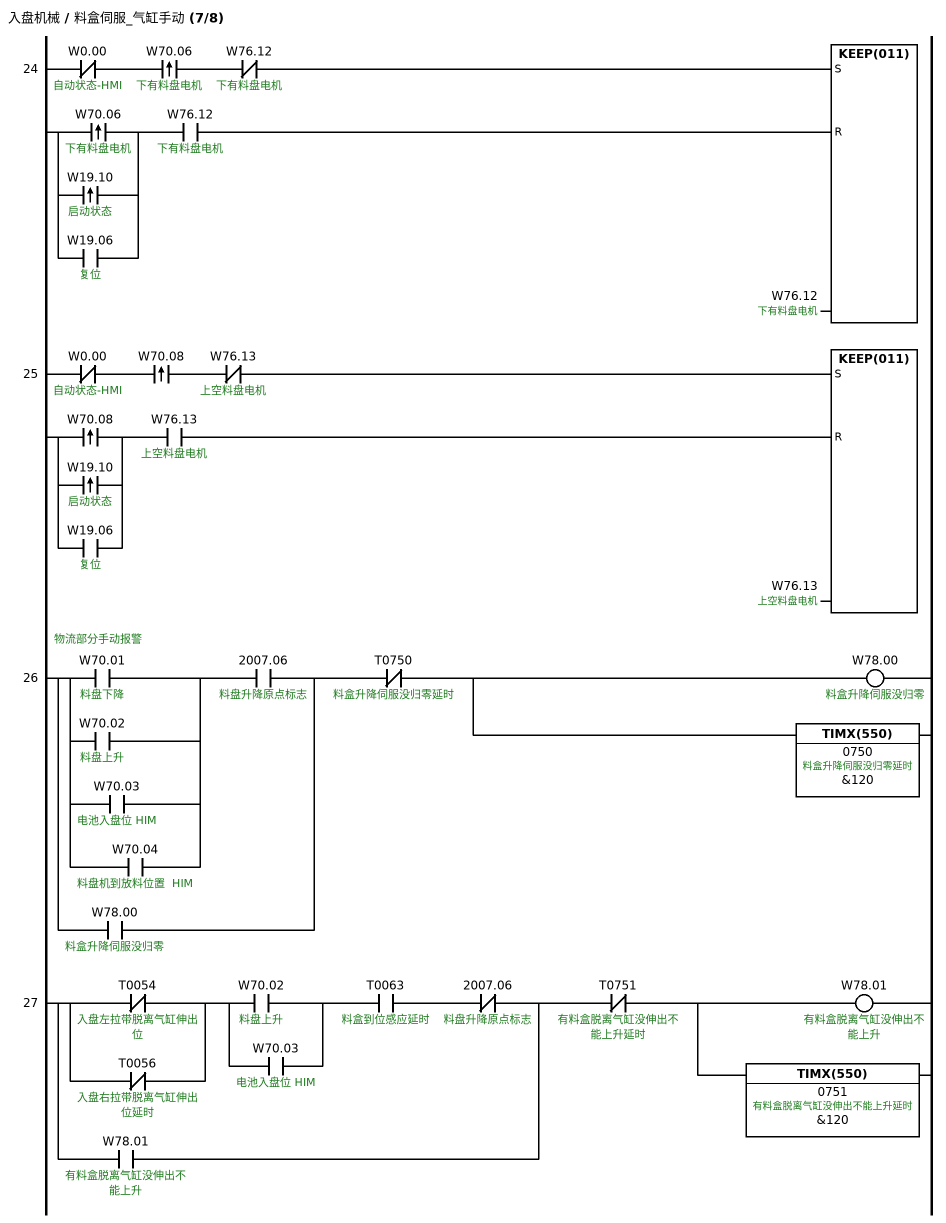
; [picture p216: 入盘机械 / 料盒伺服_气缸手动, rungs 24-27]
; rung 24
LDNOT W0.00  ; 自动状态-HMI
@AND W70.06  ; 下有料盘电机
ANDNOT W76.12  ; 下有料盘电机
@LD W70.06  ; 下有料盘电机
@OR W19.10  ; 启动状态
OR W19.06  ; 复位
AND W76.12  ; 下有料盘电机
KEEP(011) W76.12  ; 下有料盘电机
; rung 25
LDNOT W0.00  ; 自动状态-HMI
@AND W70.08
ANDNOT W76.13  ; 上空料盘电机
@LD W70.08
@OR W19.10  ; 启动状态
OR W19.06  ; 复位
AND W76.13  ; 上空料盘电机
KEEP(011) W76.13  ; 上空料盘电机
; rung 26: 物流部分手动报警
LD W70.01  ; 料盘下降
OR W70.02  ; 料盘上升
OR W70.03  ; 电池入盘位 HIM
OR W70.04  ; 料盘机到放料位置  HIM
AND 2007.06  ; 料盘升降原点标志
OR W78.00  ; 料盒升降伺服没归零
ANDNOT T0750  ; 料盒升降伺服没归零延时
OUT W78.00  ; 料盒升降伺服没归零
TIMX(550) 0750 &120  ; 料盒升降伺服没归零延时
; rung 27
LDNOT T0054  ; 入盘左拉带脱离气缸伸出位
ORNOT T0056  ; 入盘右拉带脱离气缸伸出位延时
LD W70.02  ; 料盘上升
OR W70.03  ; 电池入盘位 HIM
ANDLD
AND T0063  ; 料盒到位感应延时
ANDNOT 2007.06  ; 料盘升降原点标志
OR W78.01  ; 有料盒脱离气缸没伸出不能上升
ANDNOT T0751  ; 有料盒脱离气缸没伸出不能上升延时
OUT W78.01  ; 有料盒脱离气缸没伸出不能上升
TIMX(550) 0751 &120  ; 有料盒脱离气缸没伸出不能上升延时

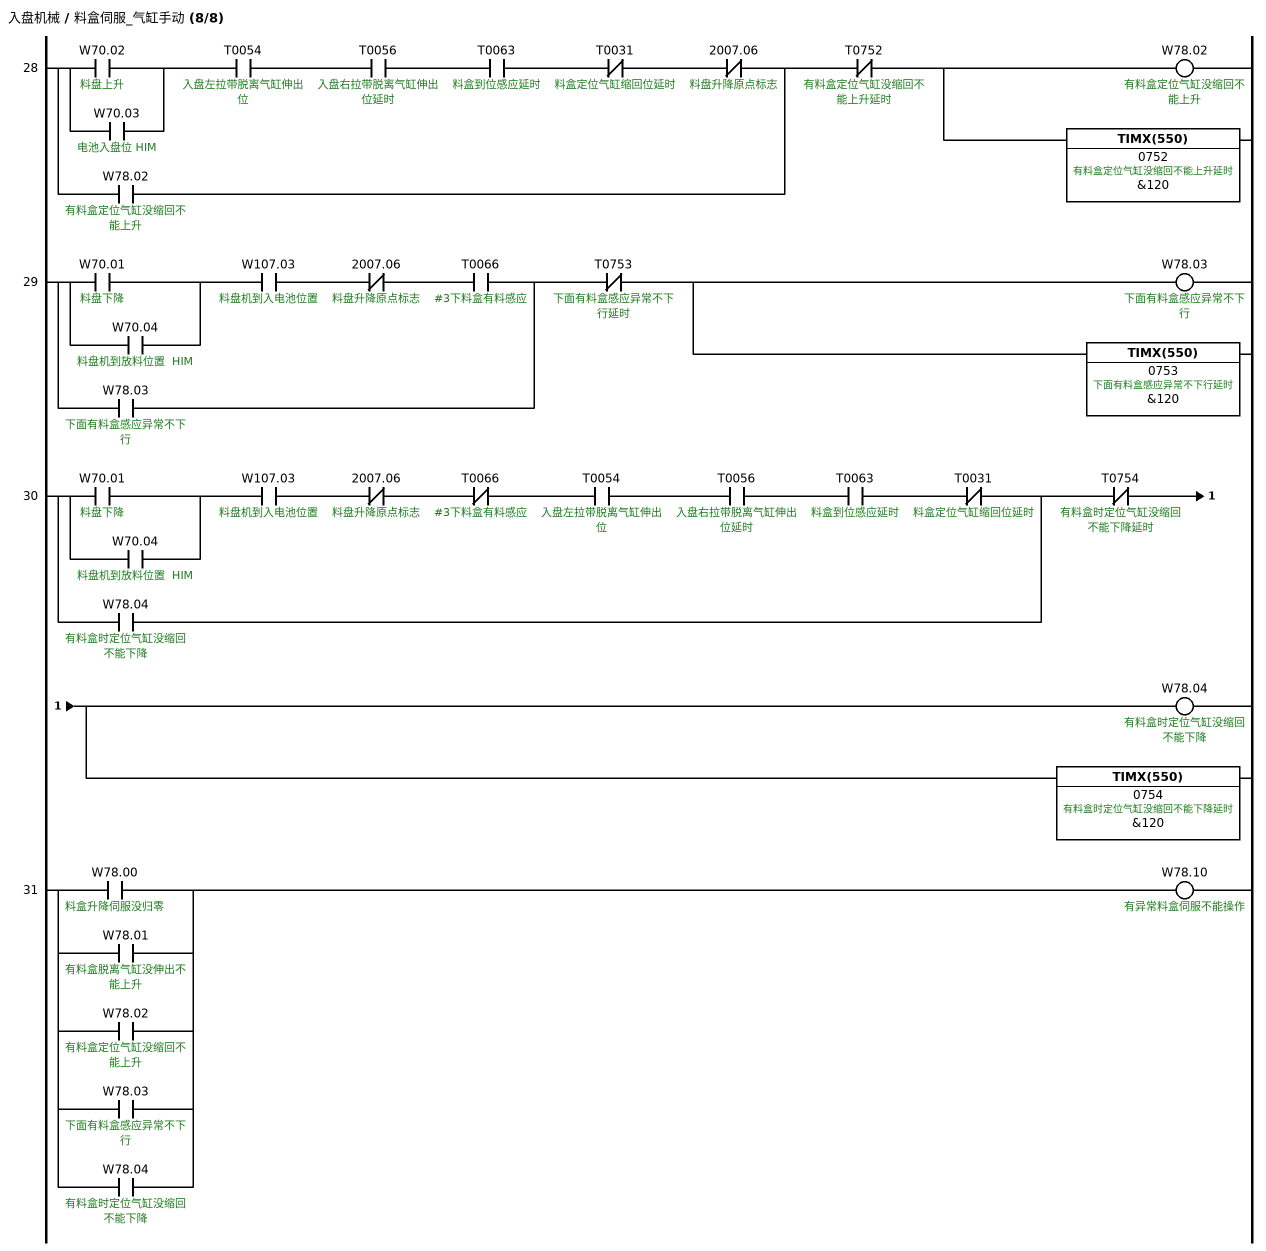
; rung 28
LD W70.02  ; 料盘上升
OR W70.03  ; 电池入盘位 HIM
AND T0054  ; 入盘左拉带脱离气缸伸出位
AND T0056  ; 入盘右拉带脱离气缸伸出位延时
AND T0063  ; 料盒到位感应延时
ANDNOT T0031  ; 料盒定位气缸缩回位延时
ANDNOT 2007.06  ; 料盘升降原点标志
OR W78.02  ; 有料盒定位气缸没缩回不能上升
ANDNOT T0752  ; 有料盒定位气缸没缩回不能上升延时
OUT W78.02  ; 有料盒定位气缸没缩回不能上升
TIMX(550) 0752 &120  ; 有料盒定位气缸没缩回不能上升延时
; rung 29
LD W70.01  ; 料盘下降
OR W70.04  ; 料盘机到放料位置  HIM
AND W107.03  ; 料盘机到入电池位置
ANDNOT 2007.06  ; 料盘升降原点标志
AND T0066  ; #3下料盒有料感应
OR W78.03  ; 下面有料盒感应异常不下行
ANDNOT T0753  ; 下面有料盒感应异常不下行延时
OUT W78.03  ; 下面有料盒感应异常不下行
TIMX(550) 0753 &120  ; 下面有料盒感应异常不下行延时
; rung 30
LD W70.01  ; 料盘下降
OR W70.04  ; 料盘机到放料位置  HIM
AND W107.03  ; 料盘机到入电池位置
ANDNOT 2007.06  ; 料盘升降原点标志
ANDNOT T0066  ; #3下料盒有料感应
AND T0054  ; 入盘左拉带脱离气缸伸出位
AND T0056  ; 入盘右拉带脱离气缸伸出位延时
AND T0063  ; 料盒到位感应延时
ANDNOT T0031  ; 料盒定位气缸缩回位延时
OR W78.04  ; 有料盒时定位气缸没缩回不能下降
ANDNOT T0754  ; 有料盒时定位气缸没缩回不能下降延时
OUT W78.04  ; 有料盒时定位气缸没缩回不能下降
TIMX(550) 0754 &120  ; 有料盒时定位气缸没缩回不能下降延时
; rung 31
LD W78.00  ; 料盒升降伺服没归零
OR W78.01  ; 有料盒脱离气缸没伸出不能上升
OR W78.02  ; 有料盒定位气缸没缩回不能上升
OR W78.03  ; 下面有料盒感应异常不下行
OR W78.04  ; 有料盒时定位气缸没缩回不能下降
OUT W78.10  ; 有异常料盒伺服不能操作

### Section 入盘自动程序

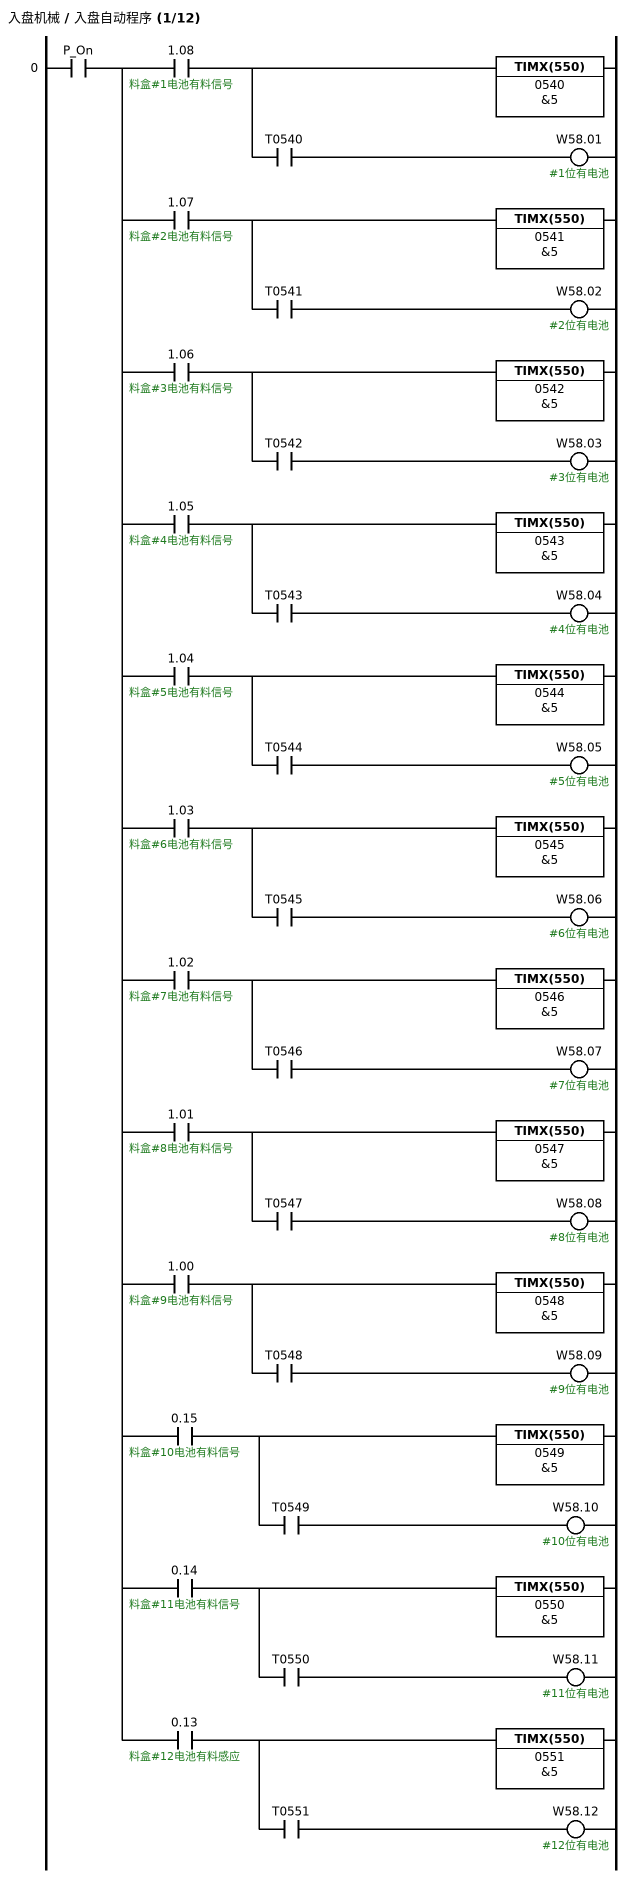
; rung 0
LD P_On
OUT TR0
AND 1.08  ; 料盒#1电池有料信号
TIMX(550) 0540 &5
AND T0540
OUT W58.01  ; #1位有电池
LD TR0
AND 1.07  ; 料盒#2电池有料信号
TIMX(550) 0541 &5
AND T0541
OUT W58.02  ; #2位有电池
LD TR0
AND 1.06  ; 料盒#3电池有料信号
TIMX(550) 0542 &5
AND T0542
OUT W58.03  ; #3位有电池
LD TR0
AND 1.05  ; 料盒#4电池有料信号
TIMX(550) 0543 &5
AND T0543
OUT W58.04  ; #4位有电池
LD TR0
AND 1.04  ; 料盒#5电池有料信号
TIMX(550) 0544 &5
AND T0544
OUT W58.05  ; #5位有电池
LD TR0
AND 1.03  ; 料盒#6电池有料信号
TIMX(550) 0545 &5
AND T0545
OUT W58.06  ; #6位有电池
LD TR0
AND 1.02  ; 料盒#7电池有料信号
TIMX(550) 0546 &5
AND T0546
OUT W58.07  ; #7位有电池
LD TR0
AND 1.01  ; 料盒#8电池有料信号
TIMX(550) 0547 &5
AND T0547
OUT W58.08  ; #8位有电池
LD TR0
AND 1.00  ; 料盒#9电池有料信号
TIMX(550) 0548 &5
AND T0548
OUT W58.09  ; #9位有电池
LD TR0
AND 0.15  ; 料盒#10电池有料信号
TIMX(550) 0549 &5
AND T0549
OUT W58.10  ; #10位有电池
LD TR0
AND 0.14  ; 料盒#11电池有料信号
TIMX(550) 0550 &5
AND T0550
OUT W58.11  ; #11位有电池
LD TR0
AND 0.13  ; 料盒#12电池有料感应
TIMX(550) 0551 &5
AND T0551
OUT W58.12  ; #12位有电池

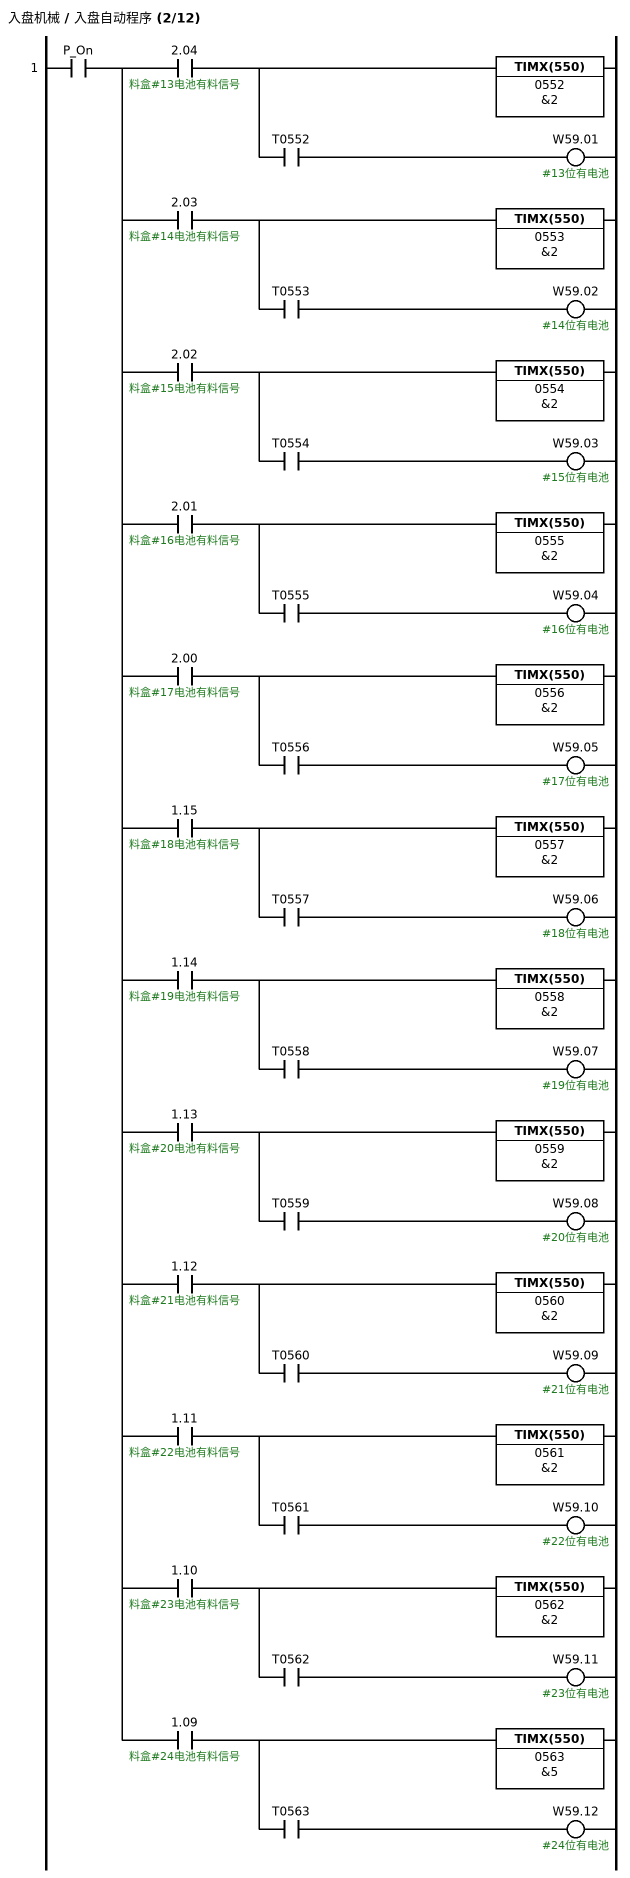
; rung 1
LD P_On
OUT TR0
AND 2.04  ; 料盒#13电池有料信号
TIMX(550) 0552 &2
AND T0552
OUT W59.01  ; #13位有电池
LD TR0
AND 2.03  ; 料盒#14电池有料信号
TIMX(550) 0553 &2
AND T0553
OUT W59.02  ; #14位有电池
LD TR0
AND 2.02  ; 料盒#15电池有料信号
TIMX(550) 0554 &2
AND T0554
OUT W59.03  ; #15位有电池
LD TR0
AND 2.01  ; 料盒#16电池有料信号
TIMX(550) 0555 &2
AND T0555
OUT W59.04  ; #16位有电池
LD TR0
AND 2.00  ; 料盒#17电池有料信号
TIMX(550) 0556 &2
AND T0556
OUT W59.05  ; #17位有电池
LD TR0
AND 1.15  ; 料盒#18电池有料信号
TIMX(550) 0557 &2
AND T0557
OUT W59.06  ; #18位有电池
LD TR0
AND 1.14  ; 料盒#19电池有料信号
TIMX(550) 0558 &2
AND T0558
OUT W59.07  ; #19位有电池
LD TR0
AND 1.13  ; 料盒#20电池有料信号
TIMX(550) 0559 &2
AND T0559
OUT W59.08  ; #20位有电池
LD TR0
AND 1.12  ; 料盒#21电池有料信号
TIMX(550) 0560 &2
AND T0560
OUT W59.09  ; #21位有电池
LD TR0
AND 1.11  ; 料盒#22电池有料信号
TIMX(550) 0561 &2
AND T0561
OUT W59.10  ; #22位有电池
LD TR0
AND 1.10  ; 料盒#23电池有料信号
TIMX(550) 0562 &2
AND T0562
OUT W59.11  ; #23位有电池
LD TR0
AND 1.09  ; 料盒#24电池有料信号
TIMX(550) 0563 &5
AND T0563
OUT W59.12  ; #24位有电池

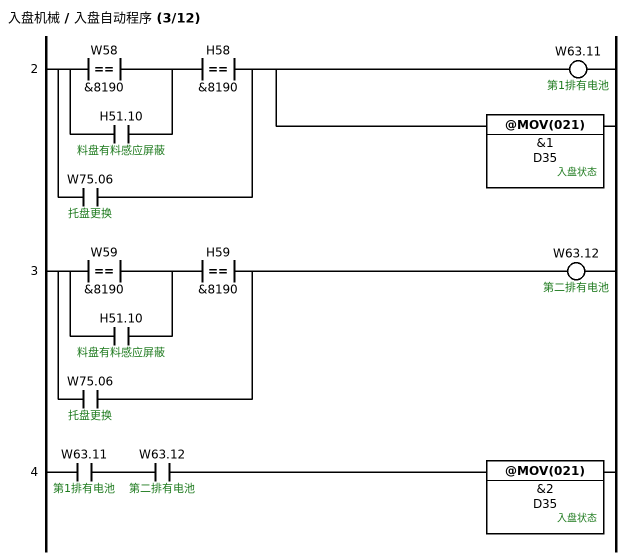
; rung 2
LD=(300) W58 &8190
OR H51.10  ; 料盘有料感应屏蔽
AND=(300) H58 &8190
OR W75.06  ; 托盘更换
OUT W63.11  ; 第1排有电池
@MOV(021) &1 D35  ; 入盘状态
; rung 3
LD=(300) W59 &8190
OR H51.10  ; 料盘有料感应屏蔽
AND=(300) H59 &8190
OR W75.06  ; 托盘更换
OUT W63.12  ; 第二排有电池
; rung 4
LD W63.11  ; 第1排有电池
AND W63.12  ; 第二排有电池
@MOV(021) &2 D35  ; 入盘状态

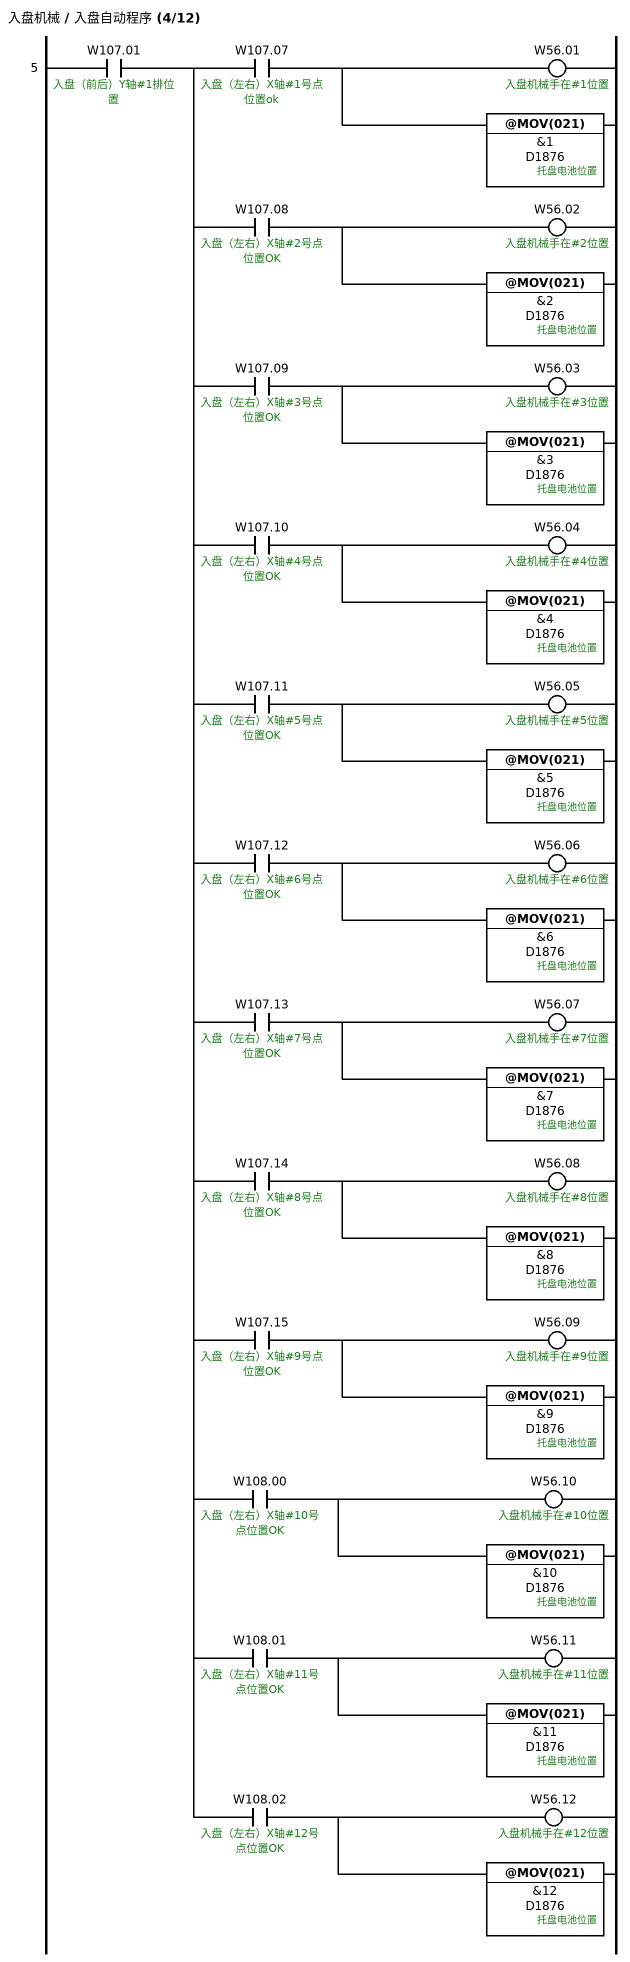
; rung 5
LD W107.01  ; 入盘（前后）Y轴#1排位置
OUT TR0
AND W107.07  ; 入盘（左右）X轴#1号点位置ok
OUT W56.01  ; 入盘机械手在#1位置
@MOV(021) &1 D1876  ; 托盘电池位置
LD TR0
AND W107.08  ; 入盘（左右）X轴#2号点位置OK
OUT W56.02  ; 入盘机械手在#2位置
@MOV(021) &2 D1876  ; 托盘电池位置
LD TR0
AND W107.09  ; 入盘（左右）X轴#3号点位置OK
OUT W56.03  ; 入盘机械手在#3位置
@MOV(021) &3 D1876  ; 托盘电池位置
LD TR0
AND W107.10  ; 入盘（左右）X轴#4号点位置OK
OUT W56.04  ; 入盘机械手在#4位置
@MOV(021) &4 D1876  ; 托盘电池位置
LD TR0
AND W107.11  ; 入盘（左右）X轴#5号点位置OK
OUT W56.05  ; 入盘机械手在#5位置
@MOV(021) &5 D1876  ; 托盘电池位置
LD TR0
AND W107.12  ; 入盘（左右）X轴#6号点位置OK
OUT W56.06  ; 入盘机械手在#6位置
@MOV(021) &6 D1876  ; 托盘电池位置
LD TR0
AND W107.13  ; 入盘（左右）X轴#7号点位置OK
OUT W56.07  ; 入盘机械手在#7位置
@MOV(021) &7 D1876  ; 托盘电池位置
LD TR0
AND W107.14  ; 入盘（左右）X轴#8号点位置OK
OUT W56.08  ; 入盘机械手在#8位置
@MOV(021) &8 D1876  ; 托盘电池位置
LD TR0
AND W107.15  ; 入盘（左右）X轴#9号点位置OK
OUT W56.09  ; 入盘机械手在#9位置
@MOV(021) &9 D1876  ; 托盘电池位置
LD TR0
AND W108.00  ; 入盘（左右）X轴#10号点位置OK
OUT W56.10  ; 入盘机械手在#10位置
@MOV(021) &10 D1876  ; 托盘电池位置
LD TR0
AND W108.01  ; 入盘（左右）X轴#11号点位置OK
OUT W56.11  ; 入盘机械手在#11位置
@MOV(021) &11 D1876  ; 托盘电池位置
LD TR0
AND W108.02  ; 入盘（左右）X轴#12号点位置OK
OUT W56.12  ; 入盘机械手在#12位置
@MOV(021) &12 D1876  ; 托盘电池位置

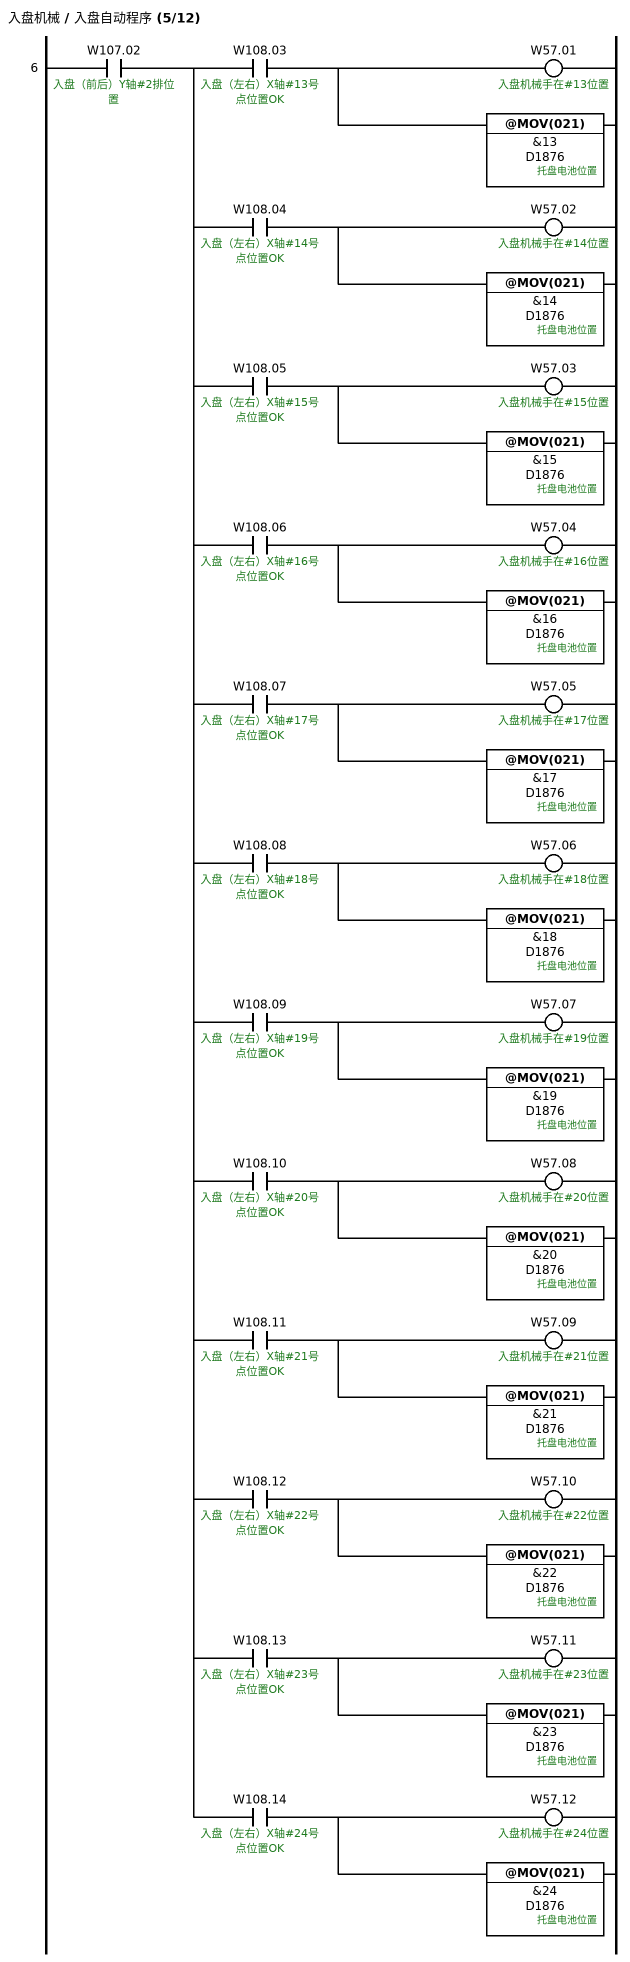
; rung 6
LD W107.02  ; 入盘（前后）Y轴#2排位置
OUT TR0
AND W108.03  ; 入盘（左右）X轴#13号点位置OK
OUT W57.01  ; 入盘机械手在#13位置
@MOV(021) &13 D1876  ; 托盘电池位置
LD TR0
AND W108.04  ; 入盘（左右）X轴#14号点位置OK
OUT W57.02  ; 入盘机械手在#14位置
@MOV(021) &14 D1876  ; 托盘电池位置
LD TR0
AND W108.05  ; 入盘（左右）X轴#15号点位置OK
OUT W57.03  ; 入盘机械手在#15位置
@MOV(021) &15 D1876  ; 托盘电池位置
LD TR0
AND W108.06  ; 入盘（左右）X轴#16号点位置OK
OUT W57.04  ; 入盘机械手在#16位置
@MOV(021) &16 D1876  ; 托盘电池位置
LD TR0
AND W108.07  ; 入盘（左右）X轴#17号点位置OK
OUT W57.05  ; 入盘机械手在#17位置
@MOV(021) &17 D1876  ; 托盘电池位置
LD TR0
AND W108.08  ; 入盘（左右）X轴#18号点位置OK
OUT W57.06  ; 入盘机械手在#18位置
@MOV(021) &18 D1876  ; 托盘电池位置
LD TR0
AND W108.09  ; 入盘（左右）X轴#19号点位置OK
OUT W57.07  ; 入盘机械手在#19位置
@MOV(021) &19 D1876  ; 托盘电池位置
LD TR0
AND W108.10  ; 入盘（左右）X轴#20号点位置OK
OUT W57.08  ; 入盘机械手在#20位置
@MOV(021) &20 D1876  ; 托盘电池位置
LD TR0
AND W108.11  ; 入盘（左右）X轴#21号点位置OK
OUT W57.09  ; 入盘机械手在#21位置
@MOV(021) &21 D1876  ; 托盘电池位置
LD TR0
AND W108.12  ; 入盘（左右）X轴#22号点位置OK
OUT W57.10  ; 入盘机械手在#22位置
@MOV(021) &22 D1876  ; 托盘电池位置
LD TR0
AND W108.13  ; 入盘（左右）X轴#23号点位置OK
OUT W57.11  ; 入盘机械手在#23位置
@MOV(021) &23 D1876  ; 托盘电池位置
LD TR0
AND W108.14  ; 入盘（左右）X轴#24号点位置OK
OUT W57.12  ; 入盘机械手在#24位置
@MOV(021) &24 D1876  ; 托盘电池位置

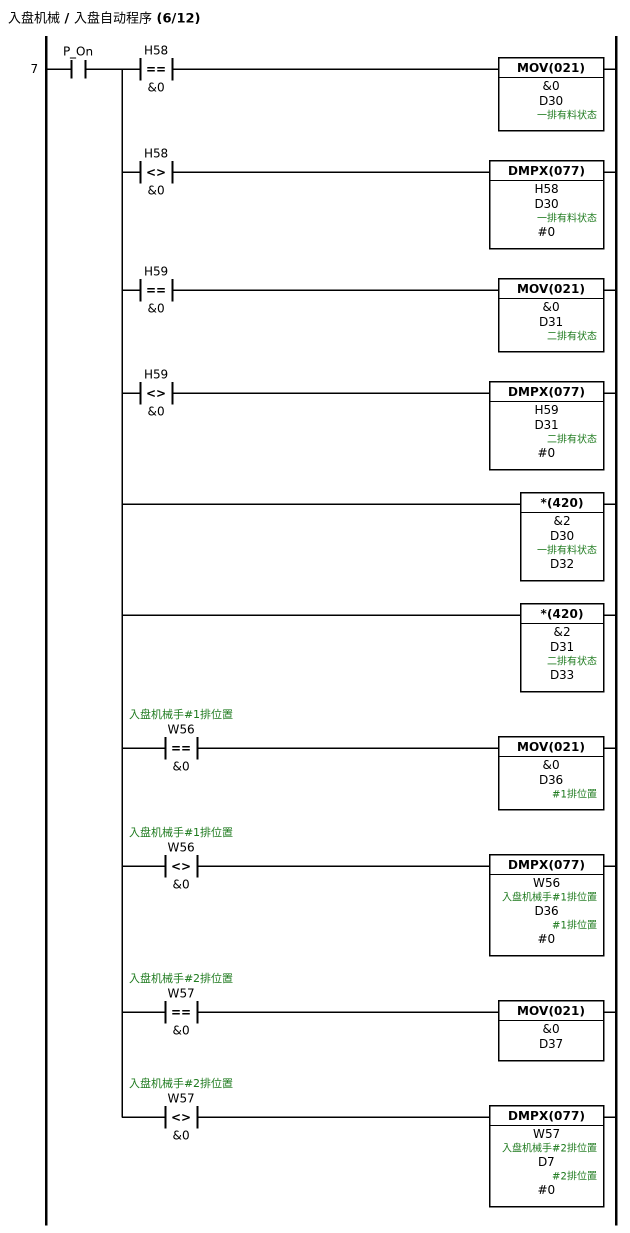
; rung 7
LD P_On
OUT TR0
AND=(300) H58 &0
MOV(021) &0 D30  ; 一排有料状态
LD TR0
AND<>(305) H58 &0
DMPX(077) H58 D30 #0  ; 一排有料状态
LD TR0
AND=(300) H59 &0
MOV(021) &0 D31  ; 二排有状态
LD TR0
AND<>(305) H59 &0
DMPX(077) H59 D31 #0  ; 二排有状态
LD TR0
*(420) &2 D30 D32  ; 一排有料状态
*(420) &2 D31 D33  ; 二排有状态
AND=(300) W56 &0  ; 入盘机械手#1排位置
MOV(021) &0 D36  ; #1排位置
LD TR0
AND<>(305) W56 &0  ; 入盘机械手#1排位置
DMPX(077) W56 D36 #0  ; 入盘机械手#1排位置, #1排位置
LD TR0
AND=(300) W57 &0  ; 入盘机械手#2排位置
MOV(021) &0 D37
LD TR0
AND<>(305) W57 &0  ; 入盘机械手#2排位置
DMPX(077) W57 D7 #0  ; 入盘机械手#2排位置, #2排位置

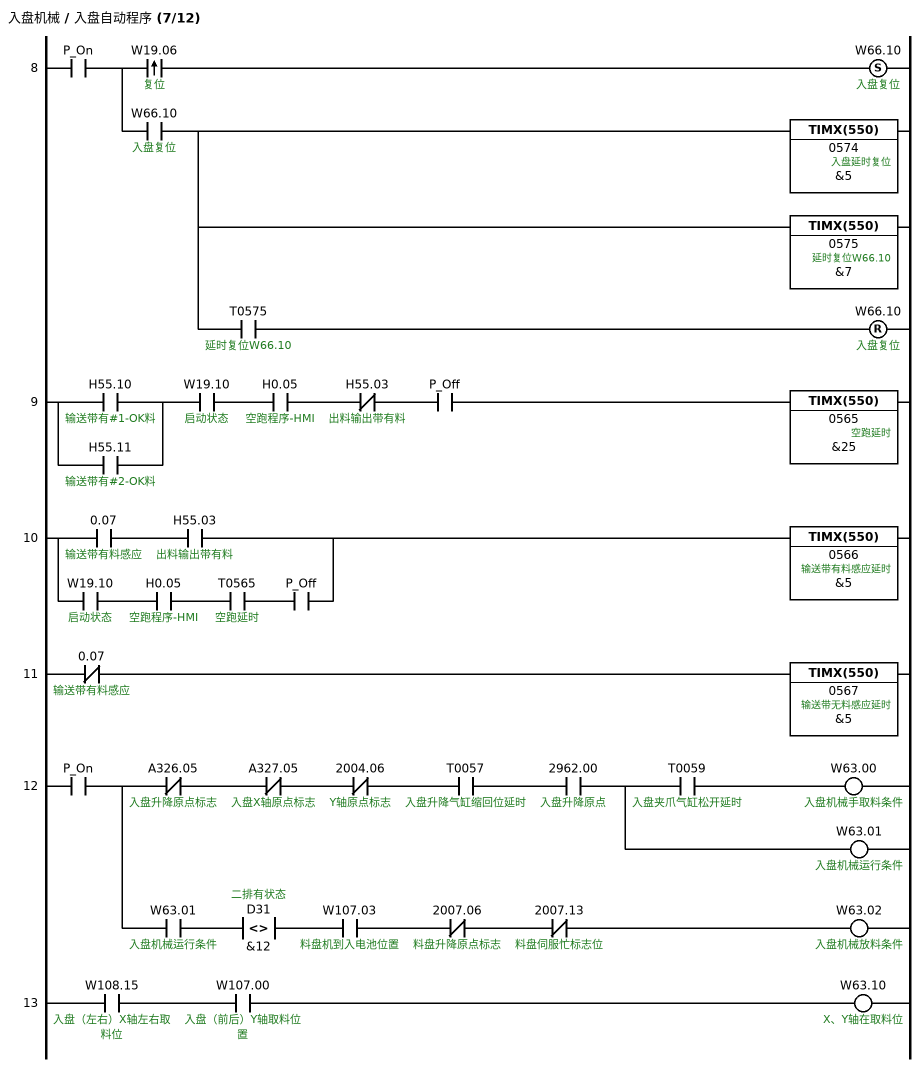
; rung 8
LD P_On
OUT TR0
@AND W19.06  ; 复位
SET W66.10  ; 入盘复位
LD TR0
AND W66.10  ; 入盘复位
TIMX(550) 0574 &5  ; 入盘延时复位
TIMX(550) 0575 &7  ; 延时复位W66.10
AND T0575  ; 延时复位W66.10
RSET W66.10  ; 入盘复位
; rung 9
LD H55.10  ; 输送带有#1-OK料
OR H55.11  ; 输送带有#2-OK料
AND W19.10  ; 启动状态
AND H0.05  ; 空跑程序-HMI
ANDNOT H55.03  ; 出料输出带有料
AND P_Off
TIMX(550) 0565 &25  ; 空跑延时
; rung 10
LD 0.07  ; 输送带有料感应
AND H55.03  ; 出料输出带有料
LD W19.10  ; 启动状态
AND H0.05  ; 空跑程序-HMI
AND T0565  ; 空跑延时
AND P_Off
ORLD
TIMX(550) 0566 &5  ; 输送带有料感应延时
; rung 11
LDNOT 0.07  ; 输送带有料感应
TIMX(550) 0567 &5  ; 输送带无料感应延时
; rung 12
LD P_On
OUT TR0
ANDNOT A326.05  ; 入盘升降原点标志
ANDNOT A327.05  ; 入盘X轴原点标志
ANDNOT 2004.06  ; Y轴原点标志
AND T0057  ; 入盘升降气缸缩回位延时
AND 2962.00  ; 入盘升降原点
OUT TR1
AND T0059  ; 入盘夹爪气缸松开延时
OUT W63.00  ; 入盘机械手取料条件
LD TR1
OUT W63.01  ; 入盘机械运行条件
LD TR0
AND W63.01  ; 入盘机械运行条件
AND<>(305) D31 &12  ; 二排有状态
AND W107.03  ; 料盘机到入电池位置
ANDNOT 2007.06  ; 料盘升降原点标志
ANDNOT 2007.13  ; 料盘伺服忙标志位
OUT W63.02  ; 入盘机械放料条件
; rung 13
LD W108.15  ; 入盘（左右）X轴左右取料位
AND W107.00  ; 入盘（前后）Y轴取料位置
OUT W63.10  ; X、Y轴在取料位

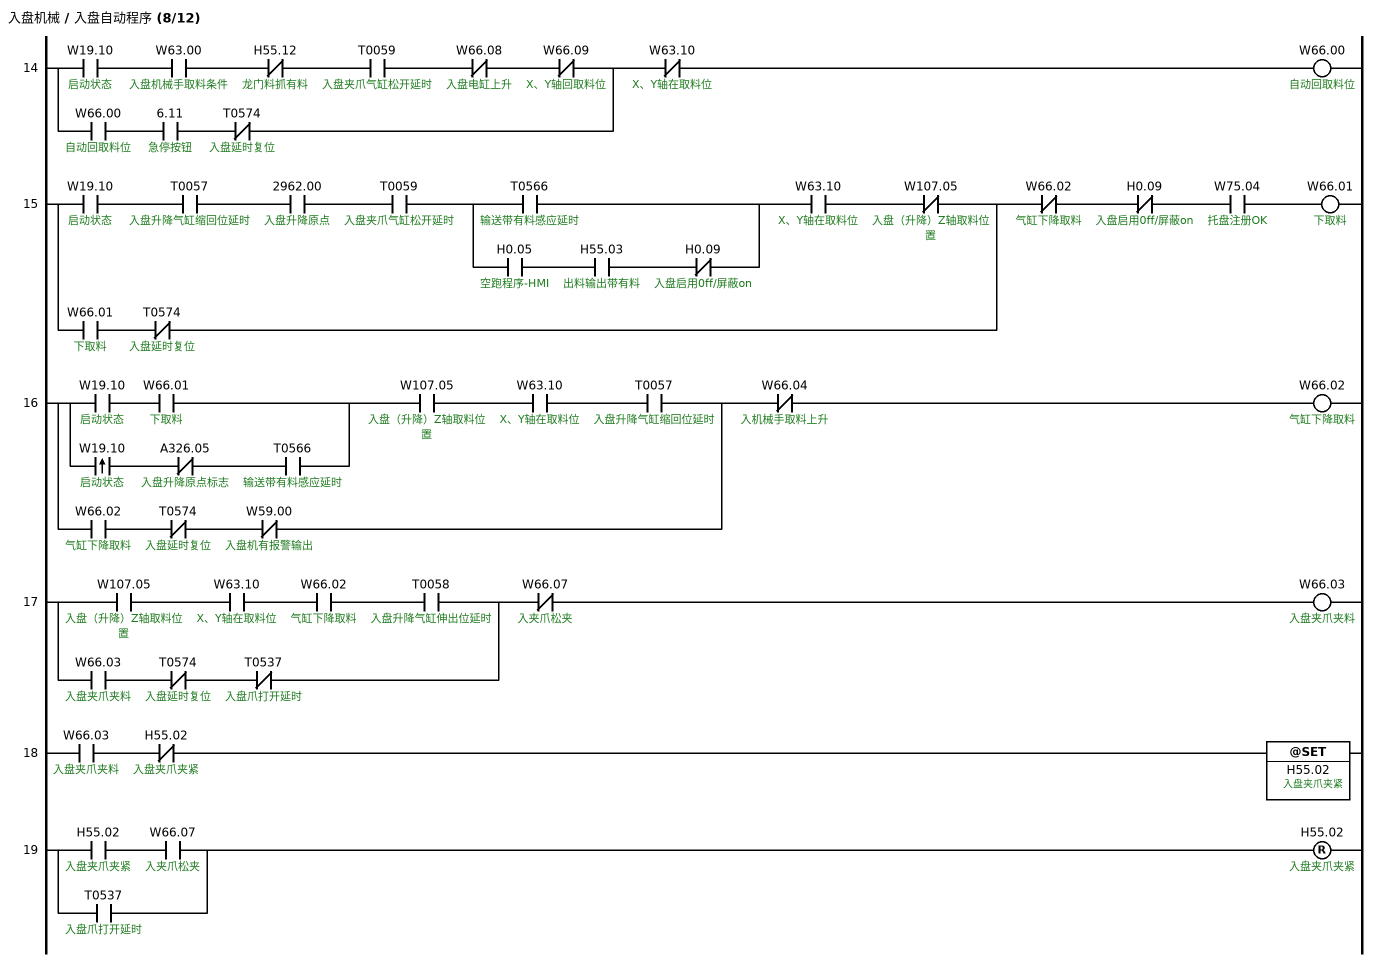
; rung 14
LD W19.10  ; 启动状态
AND W63.00  ; 入盘机械手取料条件
ANDNOT H55.12  ; 龙门料抓有料
AND T0059  ; 入盘夹爪气缸松开延时
ANDNOT W66.08  ; 入盘电缸上升
ANDNOT W66.09  ; X、Y轴回取料位
LD W66.00  ; 自动回取料位
AND 6.11  ; 急停按钮
ANDNOT T0574  ; 入盘延时复位
ORLD
ANDNOT W63.10  ; X、Y轴在取料位
OUT W66.00  ; 自动回取料位
; rung 15
LD W19.10  ; 启动状态
AND T0057  ; 入盘升降气缸缩回位延时
AND 2962.00  ; 入盘升降原点
AND T0059  ; 入盘夹爪气缸松开延时
LD T0566  ; 输送带有料感应延时
LD H0.05  ; 空跑程序-HMI
AND H55.03  ; 出料输出带有料
ANDNOT H0.09  ; 入盘启用0ff/屏蔽on
ORLD
ANDLD
AND W63.10  ; X、Y轴在取料位
ANDNOT W107.05  ; 入盘（升降）Z轴取料位置
LD W66.01  ; 下取料
ANDNOT T0574  ; 入盘延时复位
ORLD
ANDNOT W66.02  ; 气缸下降取料
ANDNOT H0.09  ; 入盘启用0ff/屏蔽on
AND W75.04  ; 托盘注册OK
OUT W66.01  ; 下取料
; rung 16
LD W19.10  ; 启动状态
AND W66.01  ; 下取料
@LD W19.10  ; 启动状态
ANDNOT A326.05  ; 入盘升降原点标志
AND T0566  ; 输送带有料感应延时
ORLD
AND W107.05  ; 入盘（升降）Z轴取料位置
AND W63.10  ; X、Y轴在取料位
AND T0057  ; 入盘升降气缸缩回位延时
LD W66.02  ; 气缸下降取料
ANDNOT T0574  ; 入盘延时复位
ANDNOT W59.00  ; 入盘机有报警输出
ORLD
ANDNOT W66.04  ; 入机械手取料上升
OUT W66.02  ; 气缸下降取料
; rung 17
LD W107.05  ; 入盘（升降）Z轴取料位置
AND W63.10  ; X、Y轴在取料位
AND W66.02  ; 气缸下降取料
AND T0058  ; 入盘升降气缸伸出位延时
LD W66.03  ; 入盘夹爪夹料
ANDNOT T0574  ; 入盘延时复位
ANDNOT T0537  ; 入盘爪打开延时
ORLD
ANDNOT W66.07  ; 入夹爪松夹
OUT W66.03  ; 入盘夹爪夹料
; rung 18
LD W66.03  ; 入盘夹爪夹料
ANDNOT H55.02  ; 入盘夹爪夹紧
@SET H55.02  ; 入盘夹爪夹紧
; rung 19
LD H55.02  ; 入盘夹爪夹紧
AND W66.07  ; 入夹爪松夹
OR T0537  ; 入盘爪打开延时
RSET H55.02  ; 入盘夹爪夹紧

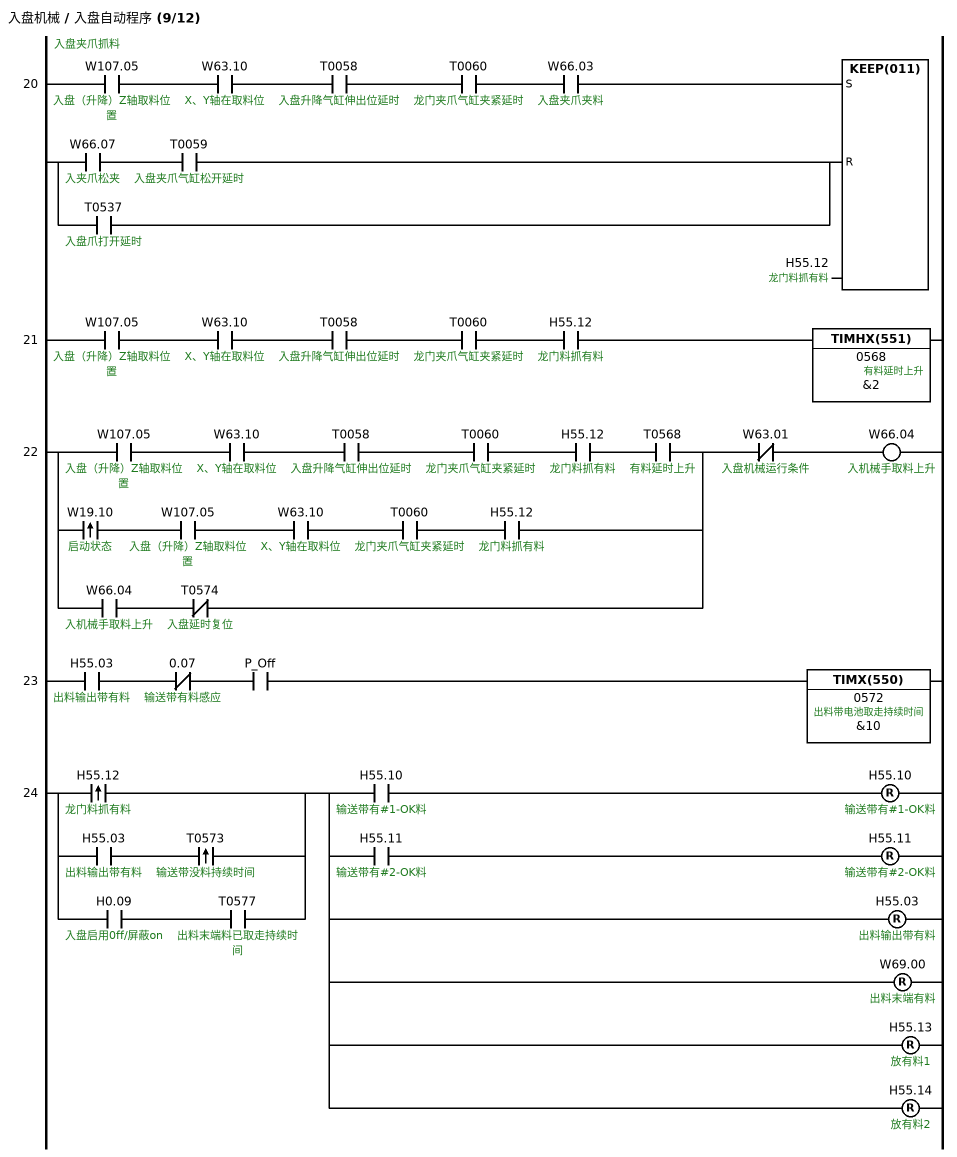
; rung 20: 入盘夹爪抓料
LD W107.05  ; 入盘（升降）Z轴取料位置
AND W63.10  ; X、Y轴在取料位
AND T0058  ; 入盘升降气缸伸出位延时
AND T0060  ; 龙门夹爪气缸夹紧延时
AND W66.03  ; 入盘夹爪夹料
LD W66.07  ; 入夹爪松夹
AND T0059  ; 入盘夹爪气缸松开延时
OR T0537  ; 入盘爪打开延时
KEEP(011) H55.12  ; 龙门料抓有料
; rung 21
LD W107.05  ; 入盘（升降）Z轴取料位置
AND W63.10  ; X、Y轴在取料位
AND T0058  ; 入盘升降气缸伸出位延时
AND T0060  ; 龙门夹爪气缸夹紧延时
AND H55.12  ; 龙门料抓有料
TIMHX(551) 0568 &2  ; 有料延时上升
; rung 22
LD W107.05  ; 入盘（升降）Z轴取料位置
AND W63.10  ; X、Y轴在取料位
AND T0058  ; 入盘升降气缸伸出位延时
AND T0060  ; 龙门夹爪气缸夹紧延时
AND H55.12  ; 龙门料抓有料
AND T0568  ; 有料延时上升
@LD W19.10  ; 启动状态
AND W107.05  ; 入盘（升降）Z轴取料位置
AND W63.10  ; X、Y轴在取料位
AND T0060  ; 龙门夹爪气缸夹紧延时
AND H55.12  ; 龙门料抓有料
ORLD
LD W66.04  ; 入机械手取料上升
ANDNOT T0574  ; 入盘延时复位
ORLD
ANDNOT W63.01  ; 入盘机械运行条件
OUT W66.04  ; 入机械手取料上升
; rung 23
LD H55.03  ; 出料输出带有料
ANDNOT 0.07  ; 输送带有料感应
AND P_Off
TIMX(550) 0572 &10  ; 出料带电池取走持续时间
; rung 24
@LD H55.12  ; 龙门料抓有料
LD H55.03  ; 出料输出带有料
@AND T0573  ; 输送带没料持续时间
ORLD
LD H0.09  ; 入盘启用0ff/屏蔽on
AND T0577  ; 出料末端料已取走持续时间
ORLD
OUT TR0
AND H55.10  ; 输送带有#1-OK料
RSET H55.10  ; 输送带有#1-OK料
LD TR0
AND H55.11  ; 输送带有#2-OK料
RSET H55.11  ; 输送带有#2-OK料
LD TR0
RSET H55.03  ; 出料输出带有料
RSET W69.00  ; 出料末端有料
RSET H55.13  ; 放有料1
RSET H55.14  ; 放有料2

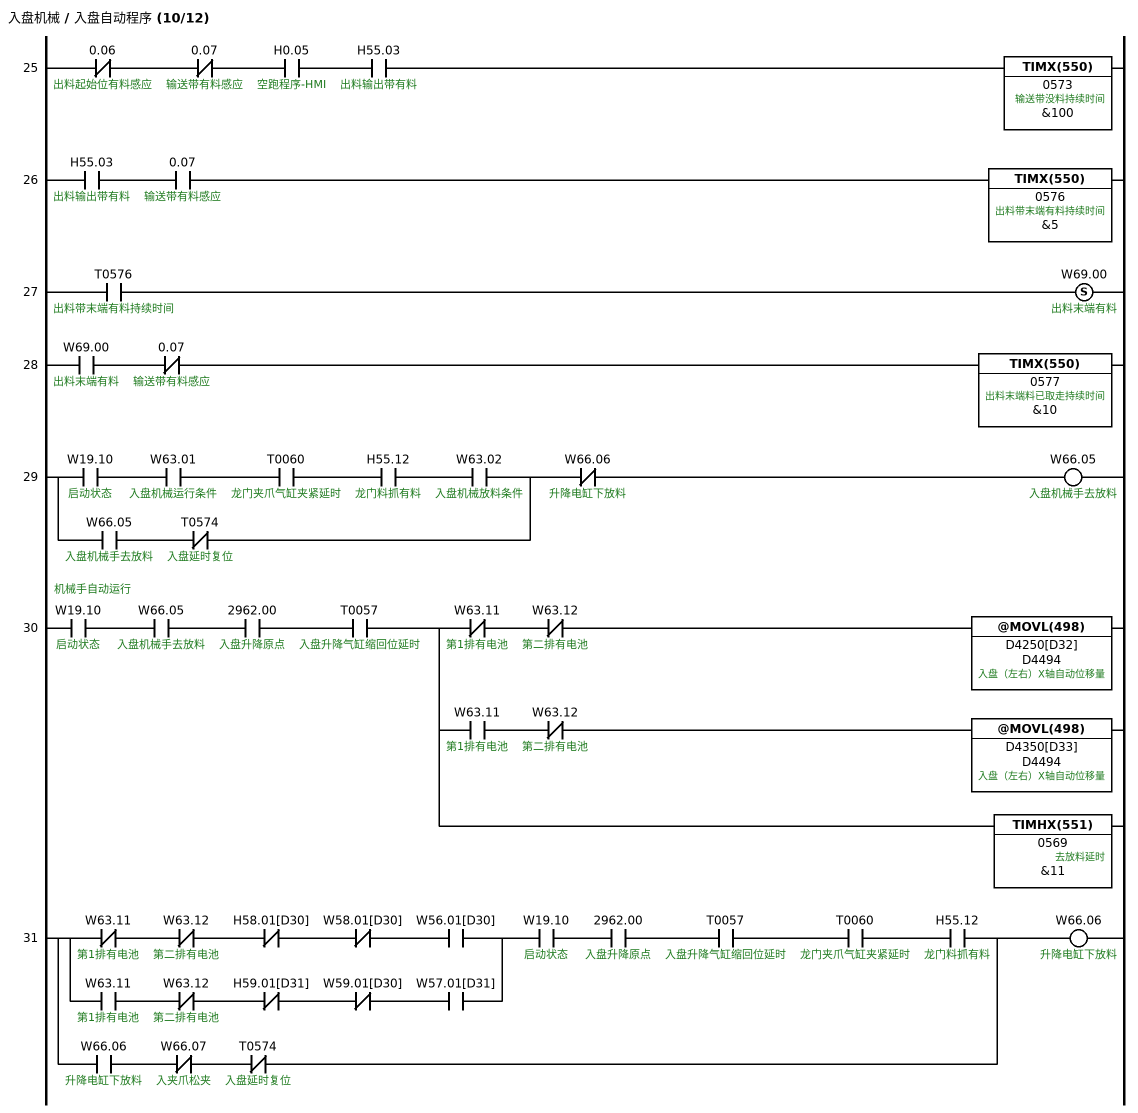
; rung 25
LDNOT 0.06  ; 出料起始位有料感应
ANDNOT 0.07  ; 输送带有料感应
AND H0.05  ; 空跑程序-HMI
AND H55.03  ; 出料输出带有料
TIMX(550) 0573 &100  ; 输送带没料持续时间
; rung 26
LD H55.03  ; 出料输出带有料
AND 0.07  ; 输送带有料感应
TIMX(550) 0576 &5  ; 出料带末端有料持续时间
; rung 27
LD T0576  ; 出料带末端有料持续时间
SET W69.00  ; 出料末端有料
; rung 28
LD W69.00  ; 出料末端有料
ANDNOT 0.07  ; 输送带有料感应
TIMX(550) 0577 &10  ; 出料末端料已取走持续时间
; rung 29
LD W19.10  ; 启动状态
AND W63.01  ; 入盘机械运行条件
AND T0060  ; 龙门夹爪气缸夹紧延时
AND H55.12  ; 龙门料抓有料
AND W63.02  ; 入盘机械放料条件
LD W66.05  ; 入盘机械手去放料
ANDNOT T0574  ; 入盘延时复位
ORLD
ANDNOT W66.06  ; 升降电缸下放料
OUT W66.05  ; 入盘机械手去放料
; rung 30: 机械手自动运行
LD W19.10  ; 启动状态
AND W66.05  ; 入盘机械手去放料
AND 2962.00  ; 入盘升降原点
AND T0057  ; 入盘升降气缸缩回位延时
OUT TR0
ANDNOT W63.11  ; 第1排有电池
ANDNOT W63.12  ; 第二排有电池
@MOVL(498) D4250[D32] D4494  ; 入盘（左右）X轴自动位移量
LD TR0
AND W63.11  ; 第1排有电池
ANDNOT W63.12  ; 第二排有电池
@MOVL(498) D4350[D33] D4494  ; 入盘（左右）X轴自动位移量
LD TR0
TIMHX(551) 0569 &11  ; 去放料延时
; rung 31
LDNOT W63.11  ; 第1排有电池
ANDNOT W63.12  ; 第二排有电池
ANDNOT H58.01[D30]
ANDNOT W58.01[D30]
AND W56.01[D30]
LD W63.11  ; 第1排有电池
ANDNOT W63.12  ; 第二排有电池
ANDNOT H59.01[D31]
ANDNOT W59.01[D30]
AND W57.01[D31]
ORLD
AND W19.10  ; 启动状态
AND 2962.00  ; 入盘升降原点
AND T0057  ; 入盘升降气缸缩回位延时
AND T0060  ; 龙门夹爪气缸夹紧延时
AND H55.12  ; 龙门料抓有料
LD W66.06  ; 升降电缸下放料
ANDNOT W66.07  ; 入夹爪松夹
ANDNOT T0574  ; 入盘延时复位
ORLD
OUT W66.06  ; 升降电缸下放料

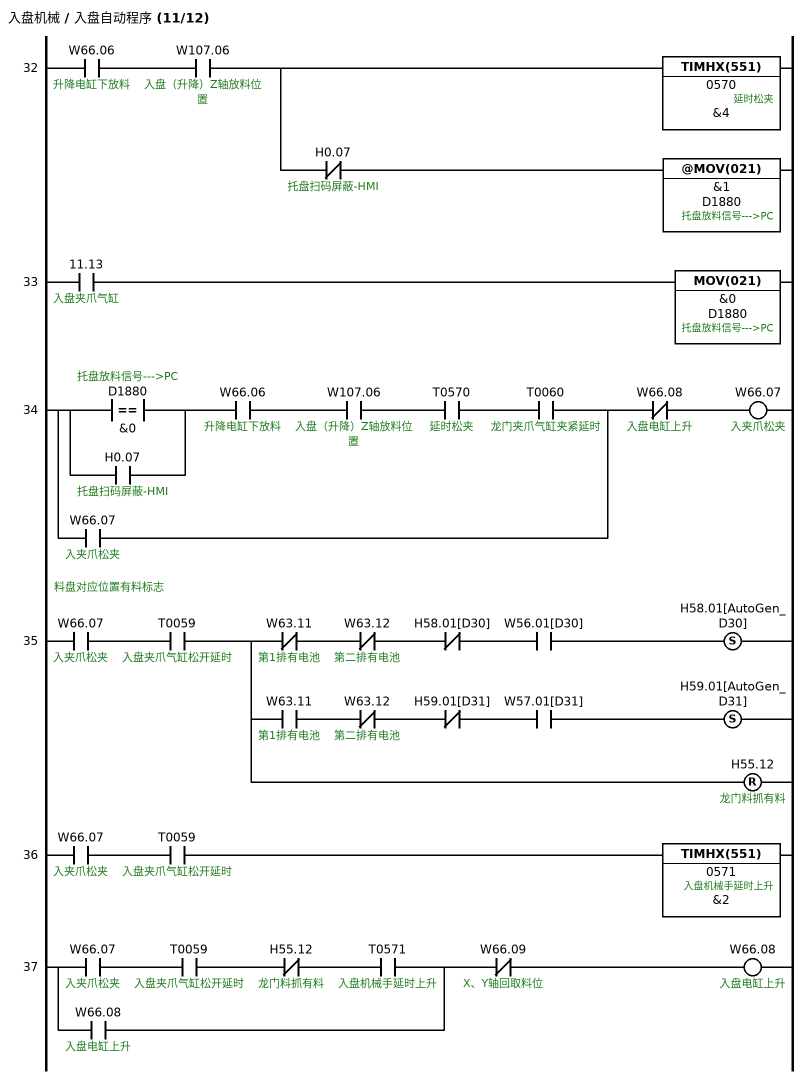
; rung 32
LD W66.06  ; 升降电缸下放料
AND W107.06  ; 入盘（升降）Z轴放料位置
TIMHX(551) 0570 &4  ; 延时松夹
ANDNOT H0.07  ; 托盘扫码屏蔽-HMI
@MOV(021) &1 D1880  ; 托盘放料信号--->PC
; rung 33
LD 11.13  ; 入盘夹爪气缸
MOV(021) &0 D1880  ; 托盘放料信号--->PC
; rung 34
LD=(300) D1880 &0  ; 托盘放料信号--->PC
OR H0.07  ; 托盘扫码屏蔽-HMI
AND W66.06  ; 升降电缸下放料
AND W107.06  ; 入盘（升降）Z轴放料位置
AND T0570  ; 延时松夹
AND T0060  ; 龙门夹爪气缸夹紧延时
OR W66.07  ; 入夹爪松夹
ANDNOT W66.08  ; 入盘电缸上升
OUT W66.07  ; 入夹爪松夹
; rung 35: 料盘对应位置有料标志
LD W66.07  ; 入夹爪松夹
AND T0059  ; 入盘夹爪气缸松开延时
OUT TR0
ANDNOT W63.11  ; 第1排有电池
ANDNOT W63.12  ; 第二排有电池
ANDNOT H58.01[D30]
AND W56.01[D30]
SET H58.01[AutoGen_D30]
LD TR0
AND W63.11  ; 第1排有电池
ANDNOT W63.12  ; 第二排有电池
ANDNOT H59.01[D31]
AND W57.01[D31]
SET H59.01[AutoGen_D31]
LD TR0
RSET H55.12  ; 龙门料抓有料
; rung 36
LD W66.07  ; 入夹爪松夹
AND T0059  ; 入盘夹爪气缸松开延时
TIMHX(551) 0571 &2  ; 入盘机械手延时上升
; rung 37
LD W66.07  ; 入夹爪松夹
AND T0059  ; 入盘夹爪气缸松开延时
ANDNOT H55.12  ; 龙门料抓有料
AND T0571  ; 入盘机械手延时上升
OR W66.08  ; 入盘电缸上升
ANDNOT W66.09  ; X、Y轴回取料位
OUT W66.08  ; 入盘电缸上升

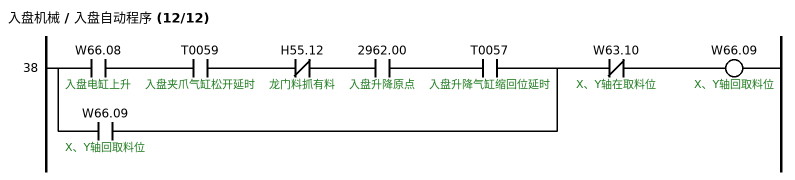
; rung 38
LD W66.08  ; 入盘电缸上升
AND T0059  ; 入盘夹爪气缸松开延时
ANDNOT H55.12  ; 龙门料抓有料
AND 2962.00  ; 入盘升降原点
AND T0057  ; 入盘升降气缸缩回位延时
OR W66.09  ; X、Y轴回取料位
ANDNOT W63.10  ; X、Y轴在取料位
OUT W66.09  ; X、Y轴回取料位

### Section 入盘自动扫码

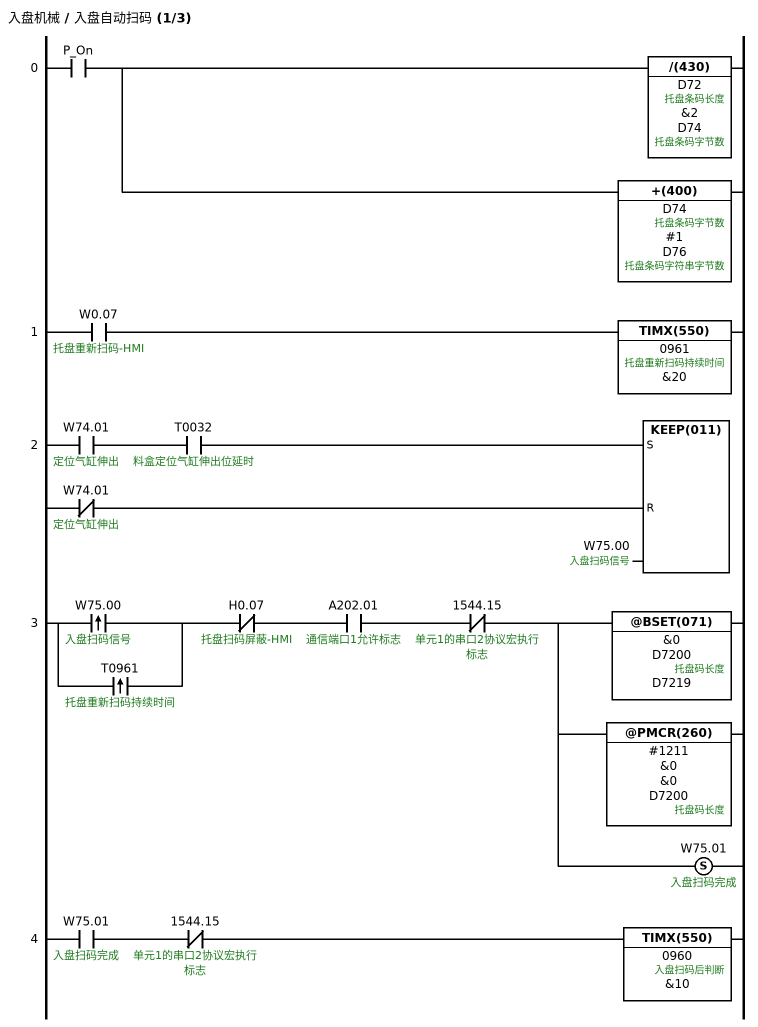
; rung 0
LD P_On
/(430) D72 &2 D74  ; 托盘条码长度, 托盘条码字节数
+(400) D74 #1 D76  ; 托盘条码字节数, 托盘条码字符串字节数
; rung 1
LD W0.07  ; 托盘重新扫码-HMI
TIMX(550) 0961 &20  ; 托盘重新扫码持续时间
; rung 2
LD W74.01  ; 定位气缸伸出
AND T0032  ; 料盒定位气缸伸出位延时
LDNOT W74.01  ; 定位气缸伸出
KEEP(011) W75.00  ; 入盘扫码信号
; rung 3
@LD W75.00  ; 入盘扫码信号
@OR T0961  ; 托盘重新扫码持续时间
ANDNOT H0.07  ; 托盘扫码屏蔽-HMI
AND A202.01  ; 通信端口1允许标志
ANDNOT 1544.15  ; 单元1的串口2协议宏执行标志
@BSET(071) &0 D7200 D7219  ; 托盘码长度
@PMCR(260) #1211 &0 &0 D7200  ; 托盘码长度
SET W75.01  ; 入盘扫码完成
; rung 4
LD W75.01  ; 入盘扫码完成
ANDNOT 1544.15  ; 单元1的串口2协议宏执行标志
TIMX(550) 0960 &10  ; 入盘扫码后判断

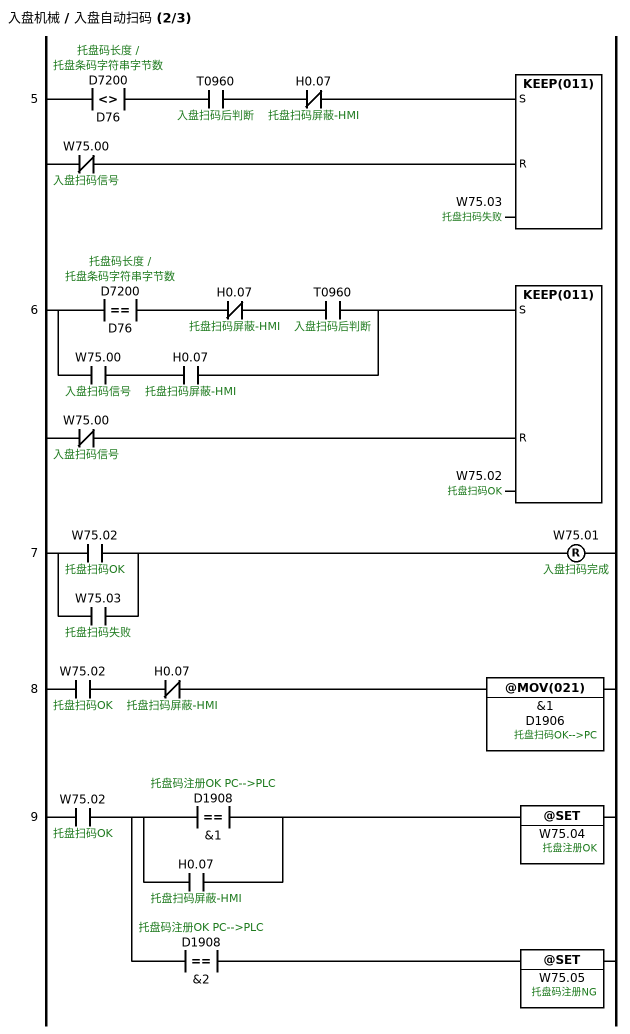
; rung 5
LD<>(305) D7200 D76  ; 托盘码长度, 托盘条码字符串字节数
AND T0960  ; 入盘扫码后判断
ANDNOT H0.07  ; 托盘扫码屏蔽-HMI
LDNOT W75.00  ; 入盘扫码信号
KEEP(011) W75.03  ; 托盘扫码失败
; rung 6
LD=(300) D7200 D76  ; 托盘码长度, 托盘条码字符串字节数
ANDNOT H0.07  ; 托盘扫码屏蔽-HMI
AND T0960  ; 入盘扫码后判断
LD W75.00  ; 入盘扫码信号
AND H0.07  ; 托盘扫码屏蔽-HMI
ORLD
LDNOT W75.00  ; 入盘扫码信号
KEEP(011) W75.02  ; 托盘扫码OK
; rung 7
LD W75.02  ; 托盘扫码OK
OR W75.03  ; 托盘扫码失败
RSET W75.01  ; 入盘扫码完成
; rung 8
LD W75.02  ; 托盘扫码OK
ANDNOT H0.07  ; 托盘扫码屏蔽-HMI
@MOV(021) &1 D1906  ; 托盘扫码OK-->PC
; rung 9
LD W75.02  ; 托盘扫码OK
OUT TR0
LD=(300) D1908 &1  ; 托盘码注册OK PC-->PLC
OR H0.07  ; 托盘扫码屏蔽-HMI
ANDLD
@SET W75.04  ; 托盘注册OK
LD TR0
AND=(300) D1908 &2  ; 托盘码注册OK PC-->PLC
@SET W75.05  ; 托盘码注册NG

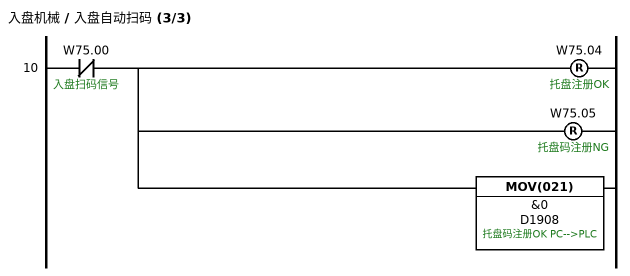
; rung 10
LDNOT W75.00  ; 入盘扫码信号
RSET W75.04  ; 托盘注册OK
RSET W75.05  ; 托盘码注册NG
MOV(021) &0 D1908  ; 托盘码注册OK PC-->PLC

### Section 入盘物流自动程序

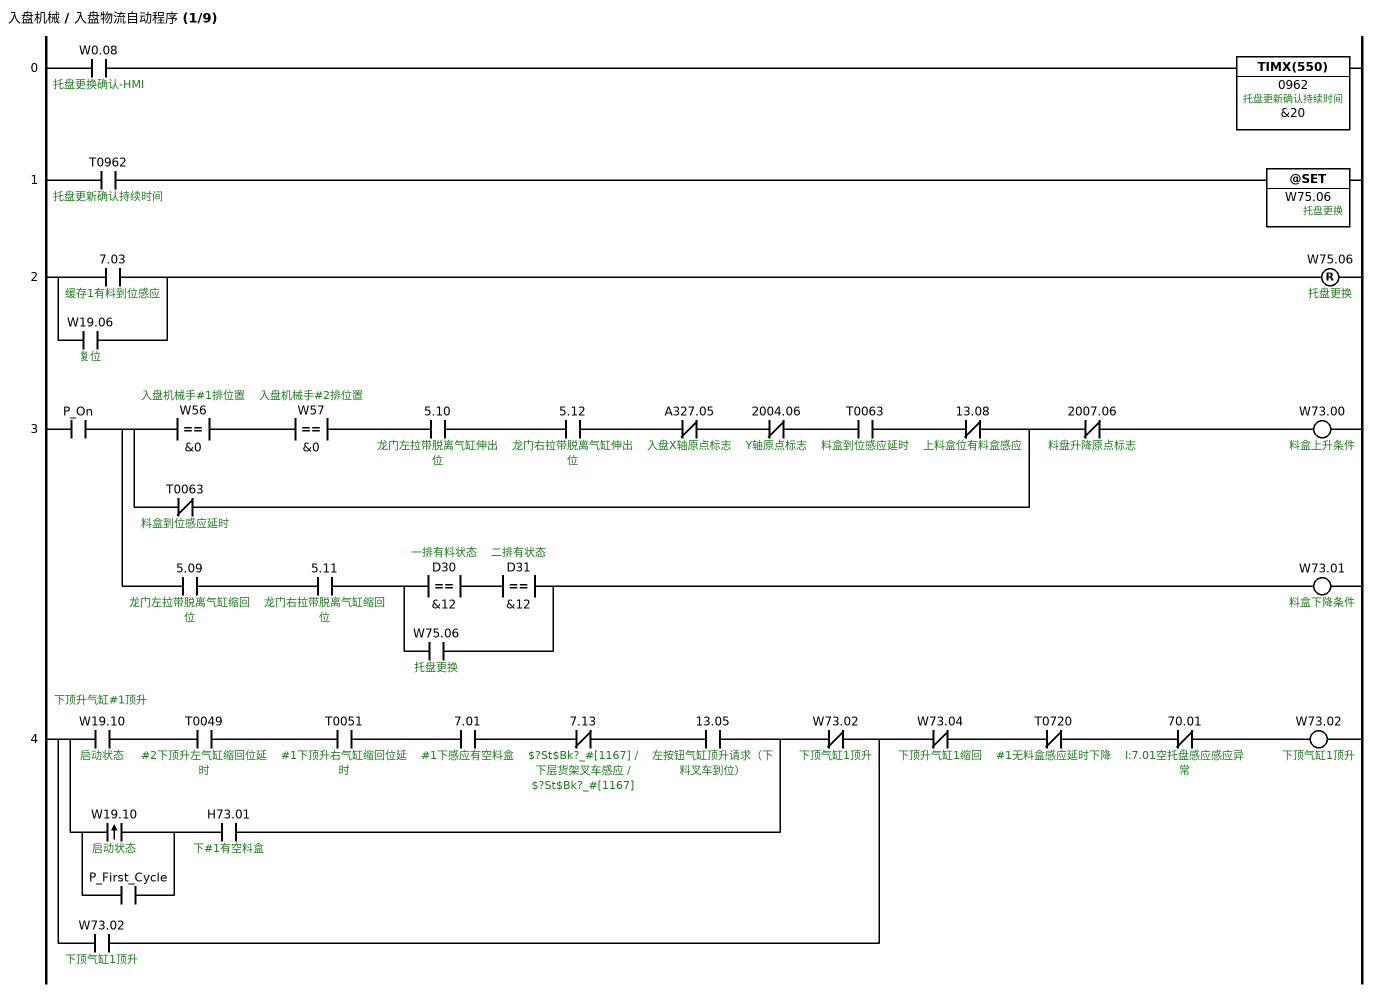
; rung 0
LD W0.08  ; 托盘更换确认-HMI
TIMX(550) 0962 &20  ; 托盘更新确认持续时间
; rung 1
LD T0962  ; 托盘更新确认持续时间
@SET W75.06  ; 托盘更换
; rung 2
LD 7.03  ; 缓存1有料到位感应
OR W19.06  ; 复位
RSET W75.06  ; 托盘更换
; rung 3
LD P_On
OUT TR0
LD=(300) W56 &0  ; 入盘机械手#1排位置
AND=(300) W57 &0  ; 入盘机械手#2排位置
AND 5.10  ; 龙门左拉带脱离气缸伸出位
AND 5.12  ; 龙门右拉带脱离气缸伸出位
ANDNOT A327.05  ; 入盘X轴原点标志
ANDNOT 2004.06  ; Y轴原点标志
AND T0063  ; 料盒到位感应延时
ANDNOT 13.08  ; 上料盒位有料盒感应
ORNOT T0063  ; 料盒到位感应延时
ANDLD
ANDNOT 2007.06  ; 料盘升降原点标志
OUT W73.00  ; 料盒上升条件
LD TR0
AND 5.09  ; 龙门左拉带脱离气缸缩回位
AND 5.11  ; 龙门右拉带脱离气缸缩回位
LD=(300) D30 &12  ; 一排有料状态
AND=(300) D31 &12  ; 二排有状态
OR W75.06  ; 托盘更换
ANDLD
OUT W73.01  ; 料盒下降条件
; rung 4: 下顶升气缸#1顶升
LD W19.10  ; 启动状态
AND T0049  ; #2下顶升左气缸缩回位延时
AND T0051  ; #1下顶升右气缸缩回位延时
AND 7.01  ; #1下感应有空料盒
ANDNOT 7.13  ; $?St$Bk?_#[1167] / 下层货架叉车感应 / $?St$Bk?_#[1167]
AND 13.05  ; 左按钮气缸顶升请求（下料叉车到位）
@LD W19.10  ; 启动状态
OR P_First_Cycle
AND H73.01  ; 下#1有空料盒
ORLD
ANDNOT W73.02  ; 下顶气缸1顶升
OR W73.02  ; 下顶气缸1顶升
ANDNOT W73.04  ; 下顶升气缸1缩回
ANDNOT T0720  ; #1无料盒感应延时下降
ANDNOT 70.01  ; I:7.01空托盘感应感应异常
OUT W73.02  ; 下顶气缸1顶升

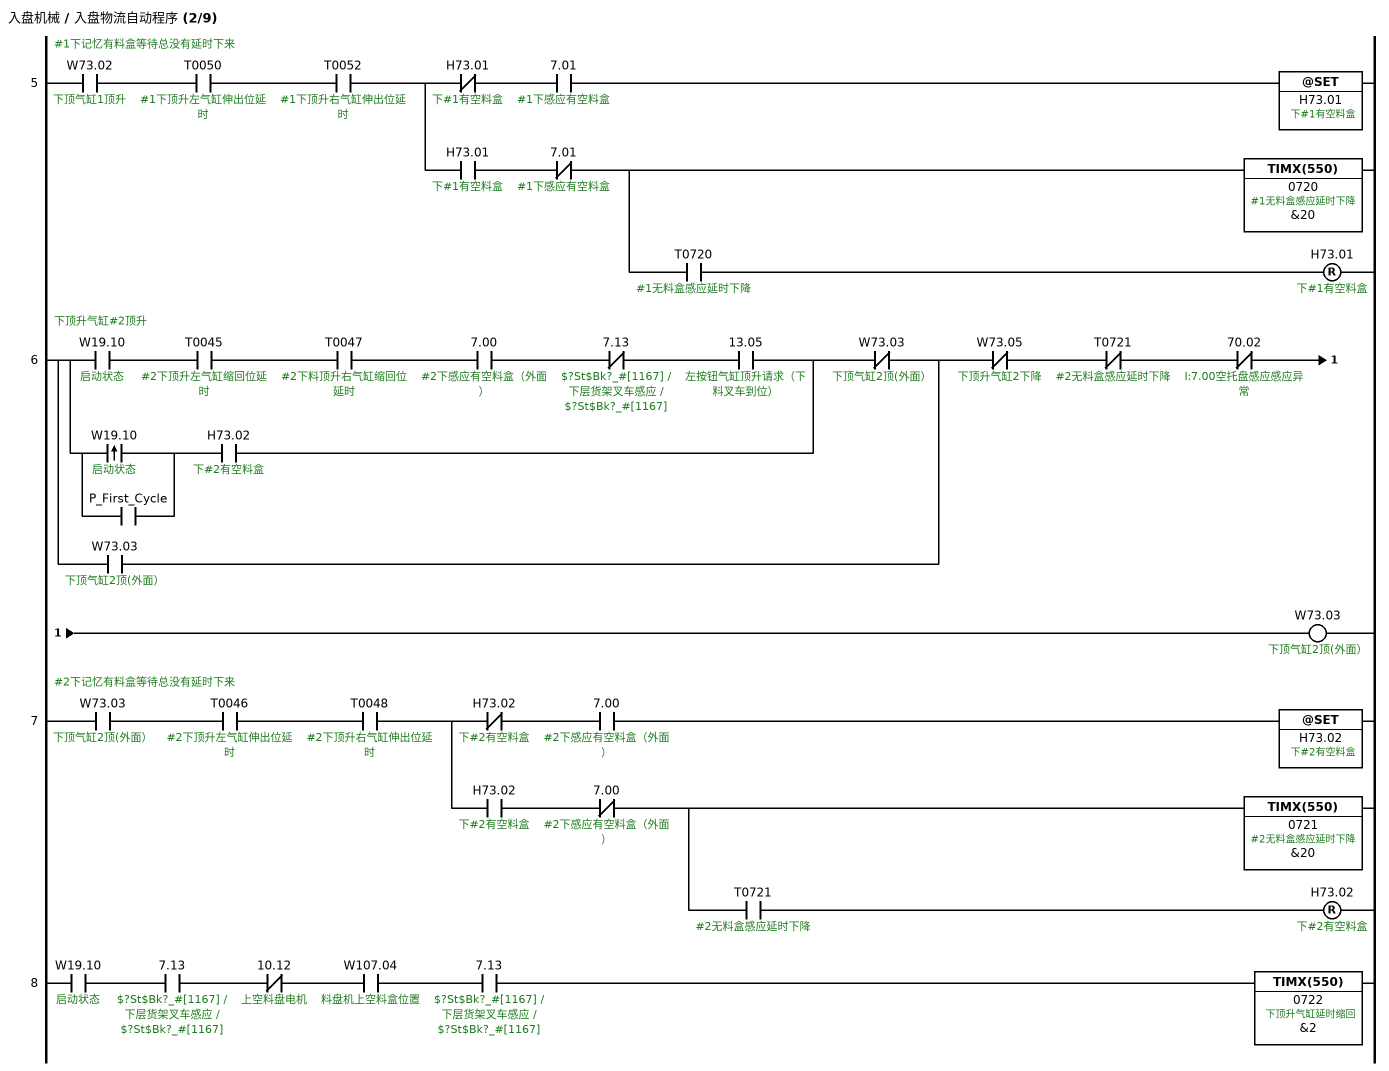
; rung 5: #1下记忆有料盒等待总没有延时下来
LD W73.02  ; 下顶气缸1顶升
AND T0050  ; #1下顶升左气缸伸出位延时
AND T0052  ; #1下顶升右气缸伸出位延时
OUT TR0
ANDNOT H73.01  ; 下#1有空料盒
AND 7.01  ; #1下感应有空料盒
@SET H73.01  ; 下#1有空料盒
LD TR0
AND H73.01  ; 下#1有空料盒
ANDNOT 7.01  ; #1下感应有空料盒
TIMX(550) 0720 &20  ; #1无料盒感应延时下降
AND T0720  ; #1无料盒感应延时下降
RSET H73.01  ; 下#1有空料盒
; rung 6: 下顶升气缸#2顶升
LD W19.10  ; 启动状态
AND T0045  ; #2下顶升左气缸缩回位延时
AND T0047  ; #2下料顶升右气缸缩回位延时
AND 7.00  ; #2下感应有空料盒（外面）
ANDNOT 7.13  ; $?St$Bk?_#[1167] / 下层货架叉车感应 / $?St$Bk?_#[1167]
AND 13.05  ; 左按钮气缸顶升请求（下料叉车到位）
@LD W19.10  ; 启动状态
OR P_First_Cycle
AND H73.02  ; 下#2有空料盒
ORLD
ANDNOT W73.03  ; 下顶气缸2顶(外面）
OR W73.03  ; 下顶气缸2顶(外面）
ANDNOT W73.05  ; 下顶升气缸2下降
ANDNOT T0721  ; #2无料盒感应延时下降
ANDNOT 70.02  ; I:7.00空托盘感应感应异常
OUT W73.03  ; 下顶气缸2顶(外面）
; rung 7: #2下记忆有料盒等待总没有延时下来
LD W73.03  ; 下顶气缸2顶(外面）
AND T0046  ; #2下顶升左气缸伸出位延时
AND T0048  ; #2下顶升右气缸伸出位延时
OUT TR0
ANDNOT H73.02  ; 下#2有空料盒
AND 7.00  ; #2下感应有空料盒（外面）
@SET H73.02  ; 下#2有空料盒
LD TR0
AND H73.02  ; 下#2有空料盒
ANDNOT 7.00  ; #2下感应有空料盒（外面）
TIMX(550) 0721 &20  ; #2无料盒感应延时下降
AND T0721  ; #2无料盒感应延时下降
RSET H73.02  ; 下#2有空料盒
; rung 8
LD W19.10  ; 启动状态
AND 7.13  ; $?St$Bk?_#[1167] / 下层货架叉车感应 / $?St$Bk?_#[1167]
ANDNOT 10.12  ; 上空料盘电机
AND W107.04  ; 料盘机上空料盒位置
AND 7.13  ; $?St$Bk?_#[1167] / 下层货架叉车感应 / $?St$Bk?_#[1167]
TIMX(550) 0722 &2  ; 下顶升气缸延时缩回

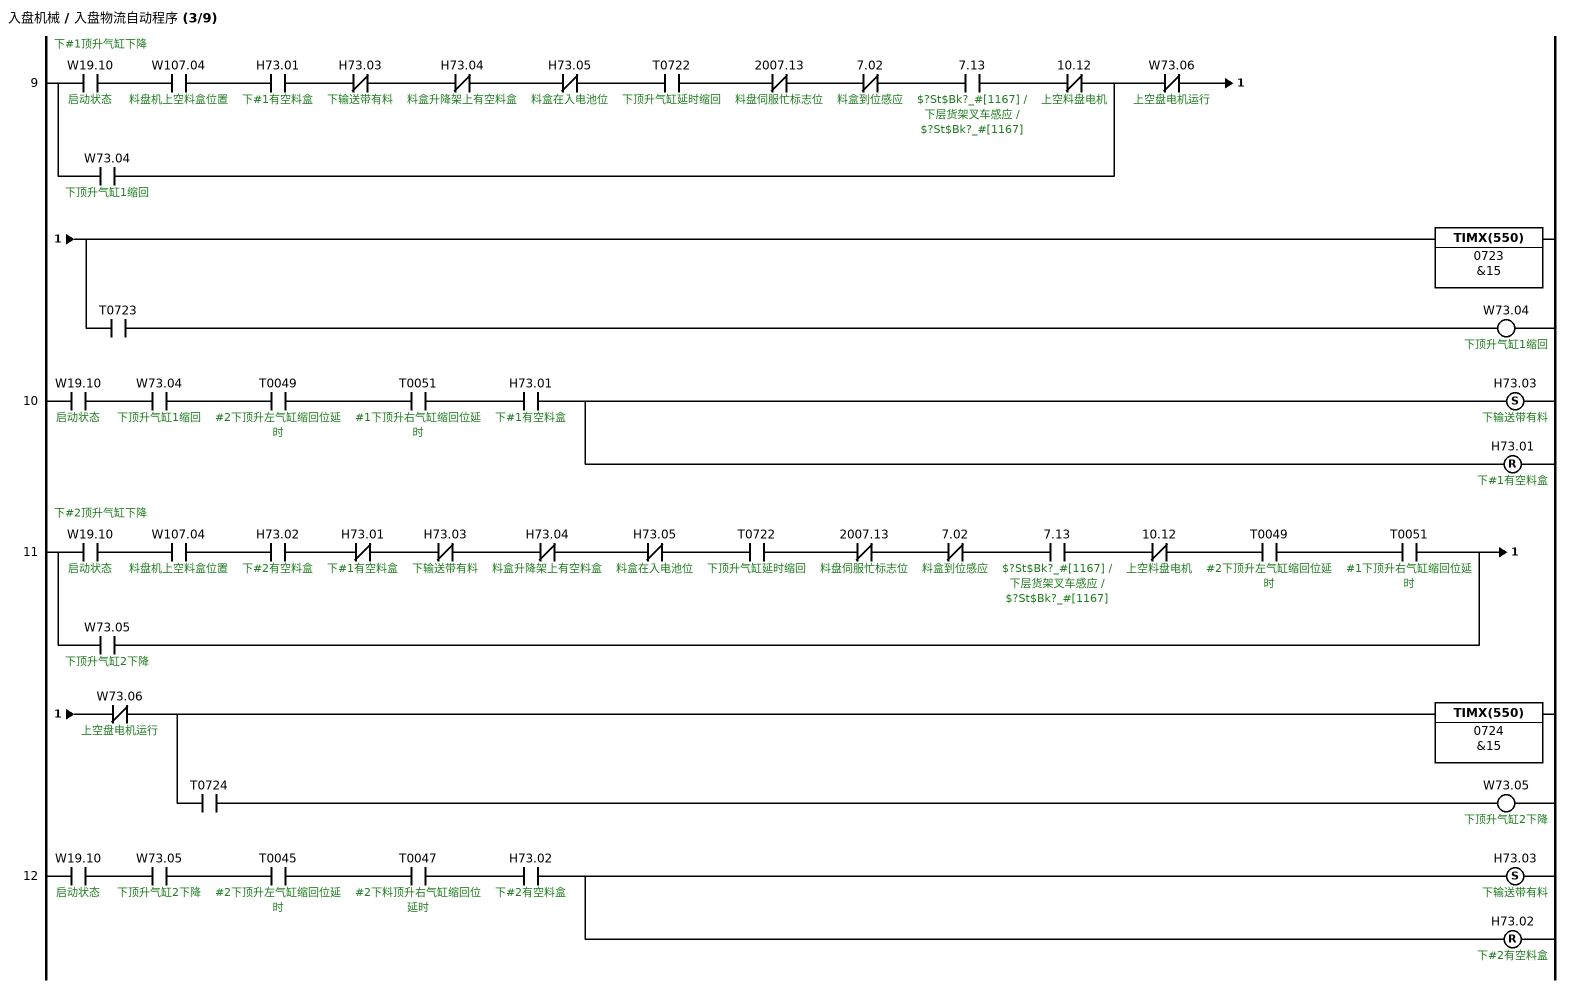
; rung 9: 下#1顶升气缸下降
LD W19.10  ; 启动状态
AND W107.04  ; 料盘机上空料盒位置
AND H73.01  ; 下#1有空料盒
ANDNOT H73.03  ; 下输送带有料
ANDNOT H73.04  ; 料盒升降架上有空料盒
ANDNOT H73.05  ; 料盒在入电池位
AND T0722  ; 下顶升气缸延时缩回
ANDNOT 2007.13  ; 料盘伺服忙标志位
ANDNOT 7.02  ; 料盒到位感应
AND 7.13  ; $?St$Bk?_#[1167] / 下层货架叉车感应 / $?St$Bk?_#[1167]
ANDNOT 10.12  ; 上空料盘电机
OR W73.04  ; 下顶升气缸1缩回
ANDNOT W73.06  ; 上空盘电机运行
TIMX(550) 0723 &15
AND T0723
OUT W73.04  ; 下顶升气缸1缩回
; rung 10
LD W19.10  ; 启动状态
AND W73.04  ; 下顶升气缸1缩回
AND T0049  ; #2下顶升左气缸缩回位延时
AND T0051  ; #1下顶升右气缸缩回位延时
AND H73.01  ; 下#1有空料盒
SET H73.03  ; 下输送带有料
RSET H73.01  ; 下#1有空料盒
; rung 11: 下#2顶升气缸下降
LD W19.10  ; 启动状态
AND W107.04  ; 料盘机上空料盒位置
AND H73.02  ; 下#2有空料盒
ANDNOT H73.01  ; 下#1有空料盒
ANDNOT H73.03  ; 下输送带有料
ANDNOT H73.04  ; 料盒升降架上有空料盒
ANDNOT H73.05  ; 料盒在入电池位
AND T0722  ; 下顶升气缸延时缩回
ANDNOT 2007.13  ; 料盘伺服忙标志位
ANDNOT 7.02  ; 料盒到位感应
AND 7.13  ; $?St$Bk?_#[1167] / 下层货架叉车感应 / $?St$Bk?_#[1167]
ANDNOT 10.12  ; 上空料盘电机
AND T0049  ; #2下顶升左气缸缩回位延时
AND T0051  ; #1下顶升右气缸缩回位延时
OR W73.05  ; 下顶升气缸2下降
ANDNOT W73.06  ; 上空盘电机运行
TIMX(550) 0724 &15
AND T0724
OUT W73.05  ; 下顶升气缸2下降
; rung 12
LD W19.10  ; 启动状态
AND W73.05  ; 下顶升气缸2下降
AND T0045  ; #2下顶升左气缸缩回位延时
AND T0047  ; #2下料顶升右气缸缩回位延时
AND H73.02  ; 下#2有空料盒
SET H73.03  ; 下输送带有料
RSET H73.02  ; 下#2有空料盒

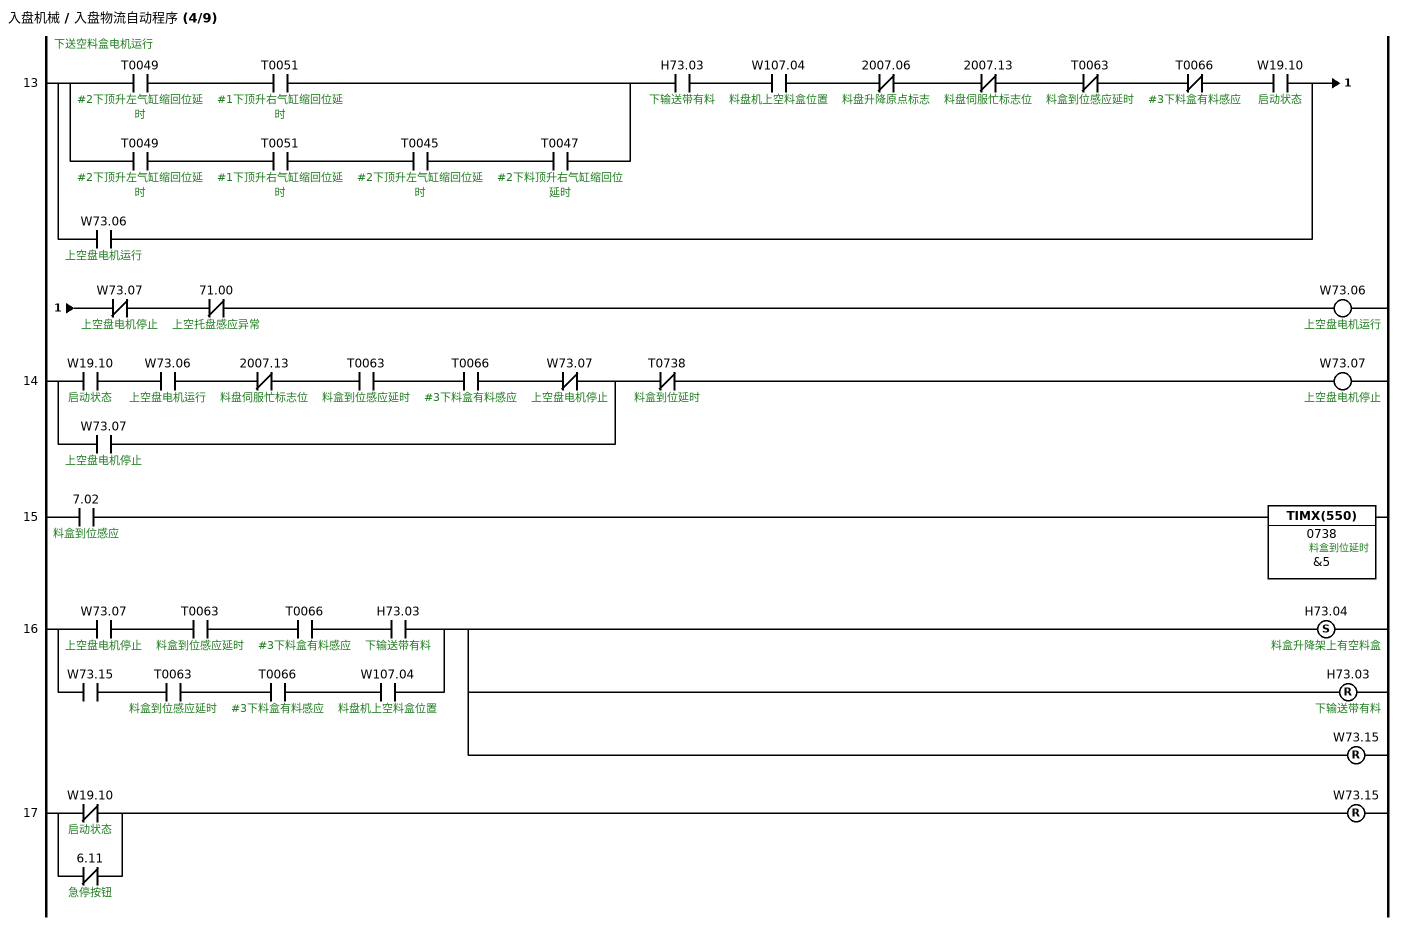
; rung 13: 下送空料盒电机运行
LD T0049  ; #2下顶升左气缸缩回位延时
AND T0051  ; #1下顶升右气缸缩回位延时
LD T0049  ; #2下顶升左气缸缩回位延时
AND T0051  ; #1下顶升右气缸缩回位延时
AND T0045  ; #2下顶升左气缸缩回位延时
AND T0047  ; #2下料顶升右气缸缩回位延时
ORLD
AND H73.03  ; 下输送带有料
AND W107.04  ; 料盘机上空料盒位置
ANDNOT 2007.06  ; 料盘升降原点标志
ANDNOT 2007.13  ; 料盘伺服忙标志位
ANDNOT T0063  ; 料盒到位感应延时
ANDNOT T0066  ; #3下料盒有料感应
AND W19.10  ; 启动状态
OR W73.06  ; 上空盘电机运行
ANDNOT W73.07  ; 上空盘电机停止
ANDNOT 71.00  ; 上空托盘感应异常
OUT W73.06  ; 上空盘电机运行
; rung 14
LD W19.10  ; 启动状态
AND W73.06  ; 上空盘电机运行
ANDNOT 2007.13  ; 料盘伺服忙标志位
AND T0063  ; 料盒到位感应延时
AND T0066  ; #3下料盒有料感应
ANDNOT W73.07  ; 上空盘电机停止
OR W73.07  ; 上空盘电机停止
ANDNOT T0738  ; 料盒到位延时
OUT W73.07  ; 上空盘电机停止
; rung 15
LD 7.02  ; 料盒到位感应
TIMX(550) 0738 &5  ; 料盒到位延时
; rung 16
LD W73.07  ; 上空盘电机停止
AND T0063  ; 料盒到位感应延时
AND T0066  ; #3下料盒有料感应
AND H73.03  ; 下输送带有料
LD W73.15
AND T0063  ; 料盒到位感应延时
AND T0066  ; #3下料盒有料感应
AND W107.04  ; 料盘机上空料盒位置
ORLD
SET H73.04  ; 料盒升降架上有空料盒
RSET H73.03  ; 下输送带有料
RSET W73.15
; rung 17
LDNOT W19.10  ; 启动状态
ORNOT 6.11  ; 急停按钮
RSET W73.15

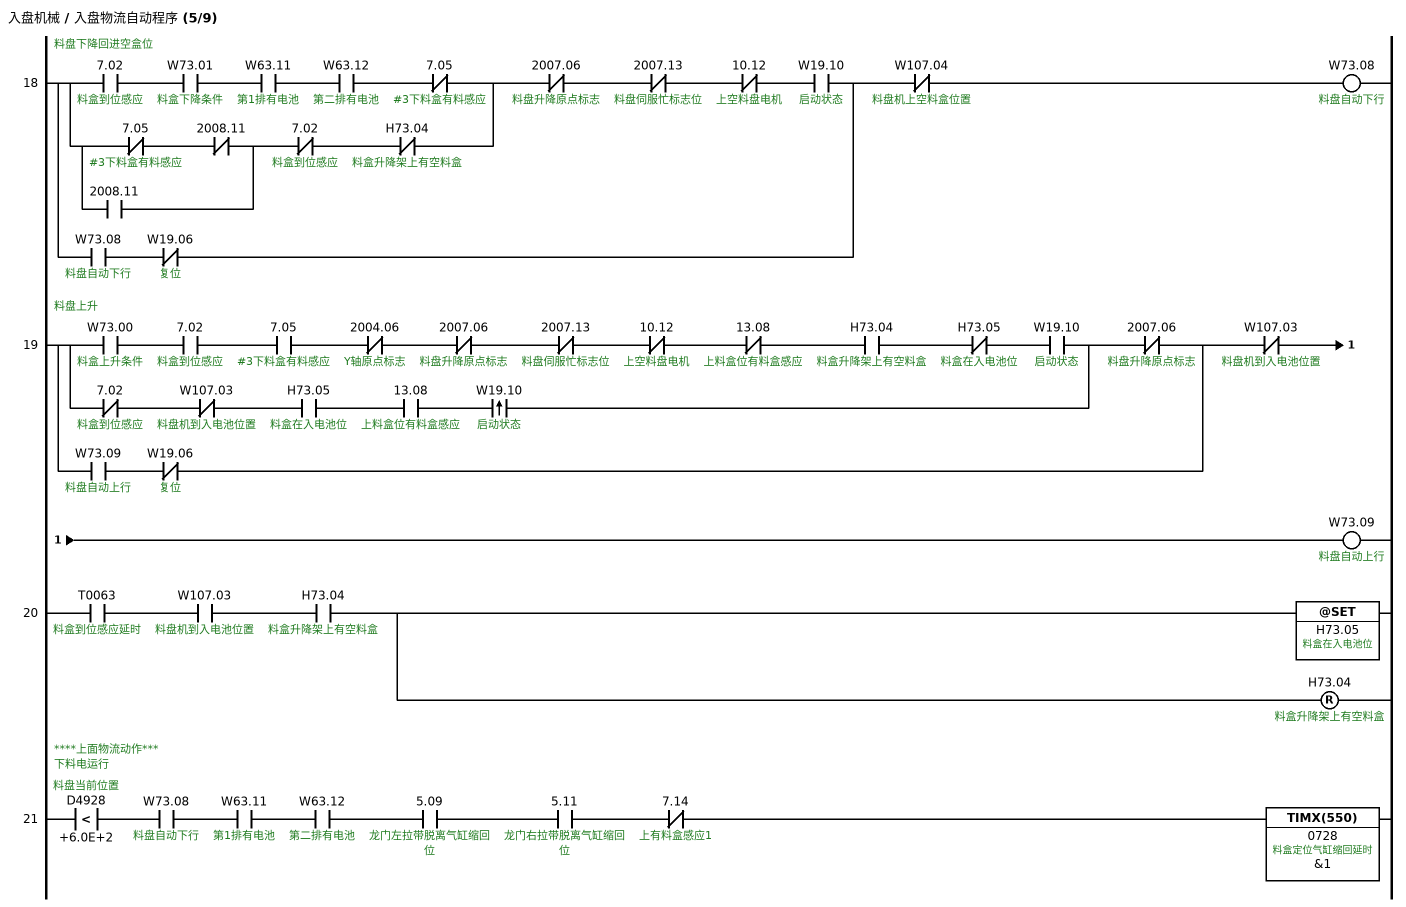
; rung 18: 料盘下降回进空盒位
LD 7.02  ; 料盒到位感应
AND W73.01  ; 料盒下降条件
AND W63.11  ; 第1排有电池
AND W63.12  ; 第二排有电池
ANDNOT 7.05  ; #3下料盒有料感应
LDNOT 7.05  ; #3下料盒有料感应
ANDNOT 2008.11
OR 2008.11
ANDNOT 7.02  ; 料盒到位感应
ANDNOT H73.04  ; 料盒升降架上有空料盒
ORLD
ANDNOT 2007.06  ; 料盘升降原点标志
ANDNOT 2007.13  ; 料盘伺服忙标志位
ANDNOT 10.12  ; 上空料盘电机
AND W19.10  ; 启动状态
LD W73.08  ; 料盘自动下行
ANDNOT W19.06  ; 复位
ORLD
ANDNOT W107.04  ; 料盘机上空料盒位置
OUT W73.08  ; 料盘自动下行
; rung 19: 料盘上升
LD W73.00  ; 料盒上升条件
AND 7.02  ; 料盒到位感应
AND 7.05  ; #3下料盒有料感应
ANDNOT 2004.06  ; Y轴原点标志
ANDNOT 2007.06  ; 料盘升降原点标志
ANDNOT 2007.13  ; 料盘伺服忙标志位
ANDNOT 10.12  ; 上空料盘电机
ANDNOT 13.08  ; 上料盒位有料盒感应
AND H73.04  ; 料盒升降架上有空料盒
ANDNOT H73.05  ; 料盒在入电池位
AND W19.10  ; 启动状态
LDNOT 7.02  ; 料盒到位感应
ANDNOT W107.03  ; 料盘机到入电池位置
AND H73.05  ; 料盒在入电池位
AND 13.08  ; 上料盒位有料盒感应
@AND W19.10  ; 启动状态
ORLD
ANDNOT 2007.06  ; 料盘升降原点标志
LD W73.09  ; 料盘自动上行
ANDNOT W19.06  ; 复位
ORLD
ANDNOT W107.03  ; 料盘机到入电池位置
OUT W73.09  ; 料盘自动上行
; rung 20
LD T0063  ; 料盒到位感应延时
AND W107.03  ; 料盘机到入电池位置
AND H73.04  ; 料盒升降架上有空料盒
@SET H73.05  ; 料盒在入电池位
RSET H73.04  ; 料盒升降架上有空料盒
; rung 21: ****上面物流动作*** / 下料电运行
LD<F(331) D4928 +6.0E+2  ; 料盘当前位置
AND W73.08  ; 料盘自动下行
AND W63.11  ; 第1排有电池
AND W63.12  ; 第二排有电池
AND 5.09  ; 龙门左拉带脱离气缸缩回位
AND 5.11  ; 龙门右拉带脱离气缸缩回位
ANDNOT 7.14  ; 上有料盒感应1
TIMX(550) 0728 &1  ; 料盒定位气缸缩回延时

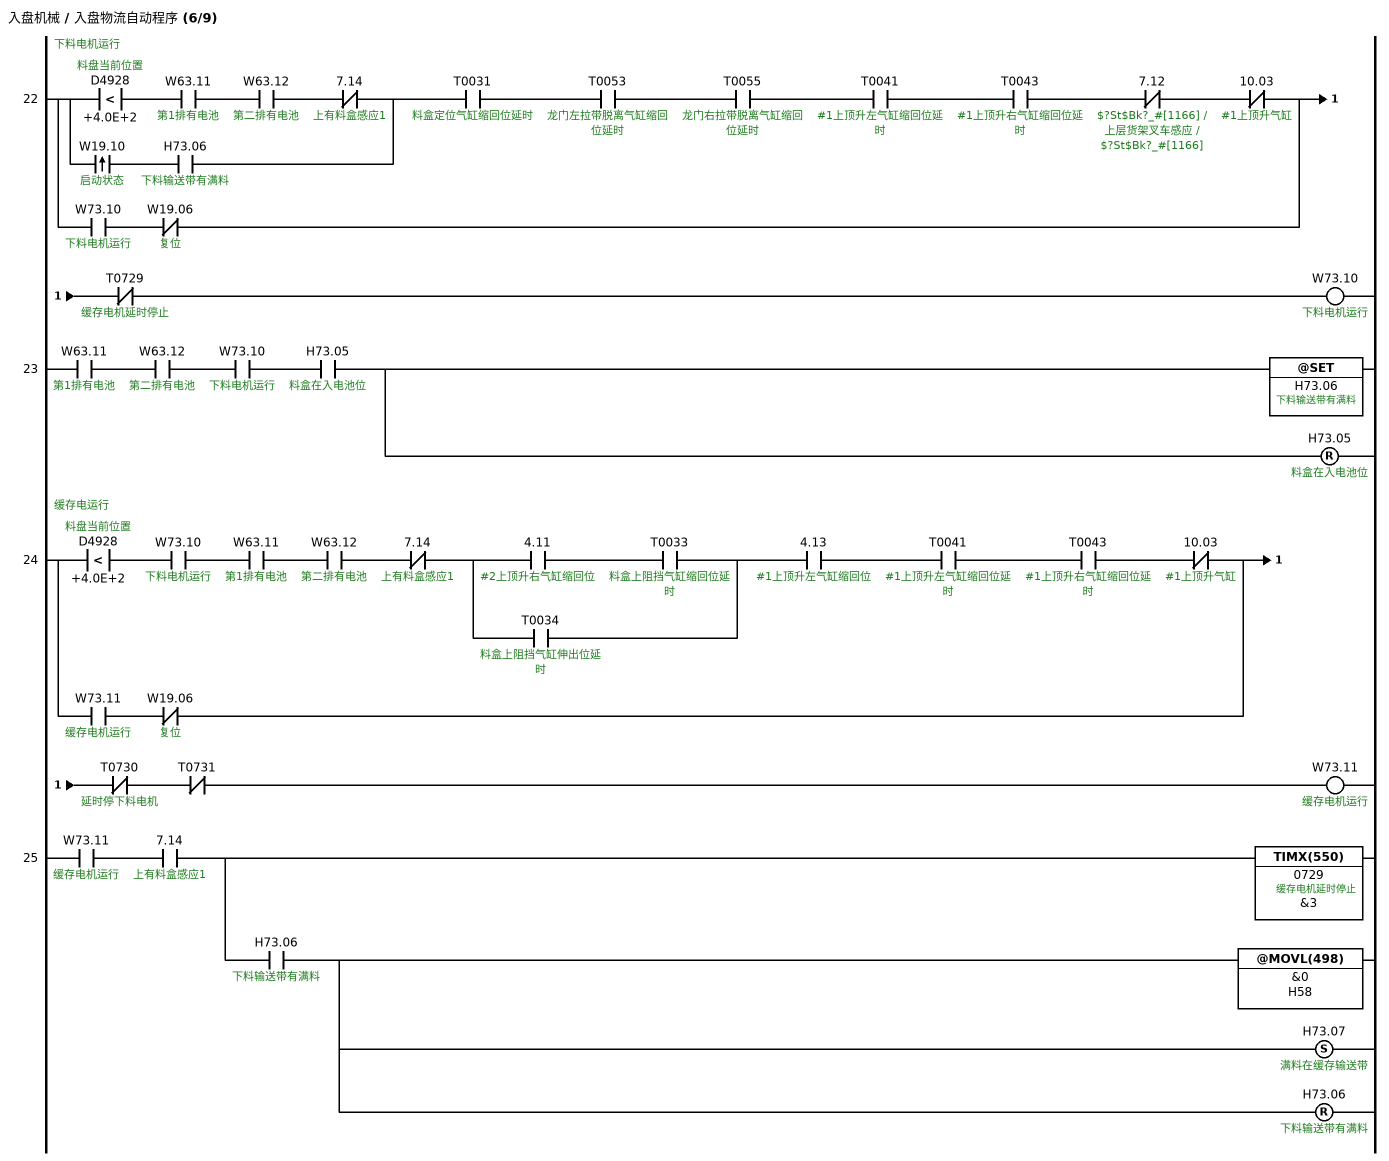
; rung 22: 下料电机运行
LD<F(331) D4928 +4.0E+2  ; 料盘当前位置
AND W63.11  ; 第1排有电池
AND W63.12  ; 第二排有电池
ANDNOT 7.14  ; 上有料盒感应1
@LD W19.10  ; 启动状态
AND H73.06  ; 下料输送带有满料
ORLD
AND T0031  ; 料盒定位气缸缩回位延时
AND T0053  ; 龙门左拉带脱离气缸缩回位延时
AND T0055  ; 龙门右拉带脱离气缸缩回位延时
AND T0041  ; #1上顶升左气缸缩回位延时
AND T0043  ; #1上顶升右气缸缩回位延时
ANDNOT 7.12  ; $?St$Bk?_#[1166] / 上层货架叉车感应 / $?St$Bk?_#[1166]
ANDNOT 10.03  ; #1上顶升气缸
LD W73.10  ; 下料电机运行
ANDNOT W19.06  ; 复位
ORLD
ANDNOT T0729  ; 缓存电机延时停止
OUT W73.10  ; 下料电机运行
; rung 23
LD W63.11  ; 第1排有电池
AND W63.12  ; 第二排有电池
AND W73.10  ; 下料电机运行
AND H73.05  ; 料盒在入电池位
@SET H73.06  ; 下料输送带有满料
RSET H73.05  ; 料盒在入电池位
; rung 24: 缓存电运行
LD<F(331) D4928 +4.0E+2  ; 料盘当前位置
AND W73.10  ; 下料电机运行
AND W63.11  ; 第1排有电池
AND W63.12  ; 第二排有电池
ANDNOT 7.14  ; 上有料盒感应1
LD 4.11  ; #2上顶升右气缸缩回位
AND T0033  ; 料盒上阻挡气缸缩回位延时
OR T0034  ; 料盒上阻挡气缸伸出位延时
ANDLD
AND 4.13  ; #1上顶升左气缸缩回位
AND T0041  ; #1上顶升左气缸缩回位延时
AND T0043  ; #1上顶升右气缸缩回位延时
ANDNOT 10.03  ; #1上顶升气缸
LD W73.11  ; 缓存电机运行
ANDNOT W19.06  ; 复位
ORLD
ANDNOT T0730  ; 延时停下料电机
ANDNOT T0731
OUT W73.11  ; 缓存电机运行
; rung 25
LD W73.11  ; 缓存电机运行
AND 7.14  ; 上有料盒感应1
TIMX(550) 0729 &3  ; 缓存电机延时停止
AND H73.06  ; 下料输送带有满料
@MOVL(498) &0 H58
SET H73.07  ; 满料在缓存输送带
RSET H73.06  ; 下料输送带有满料

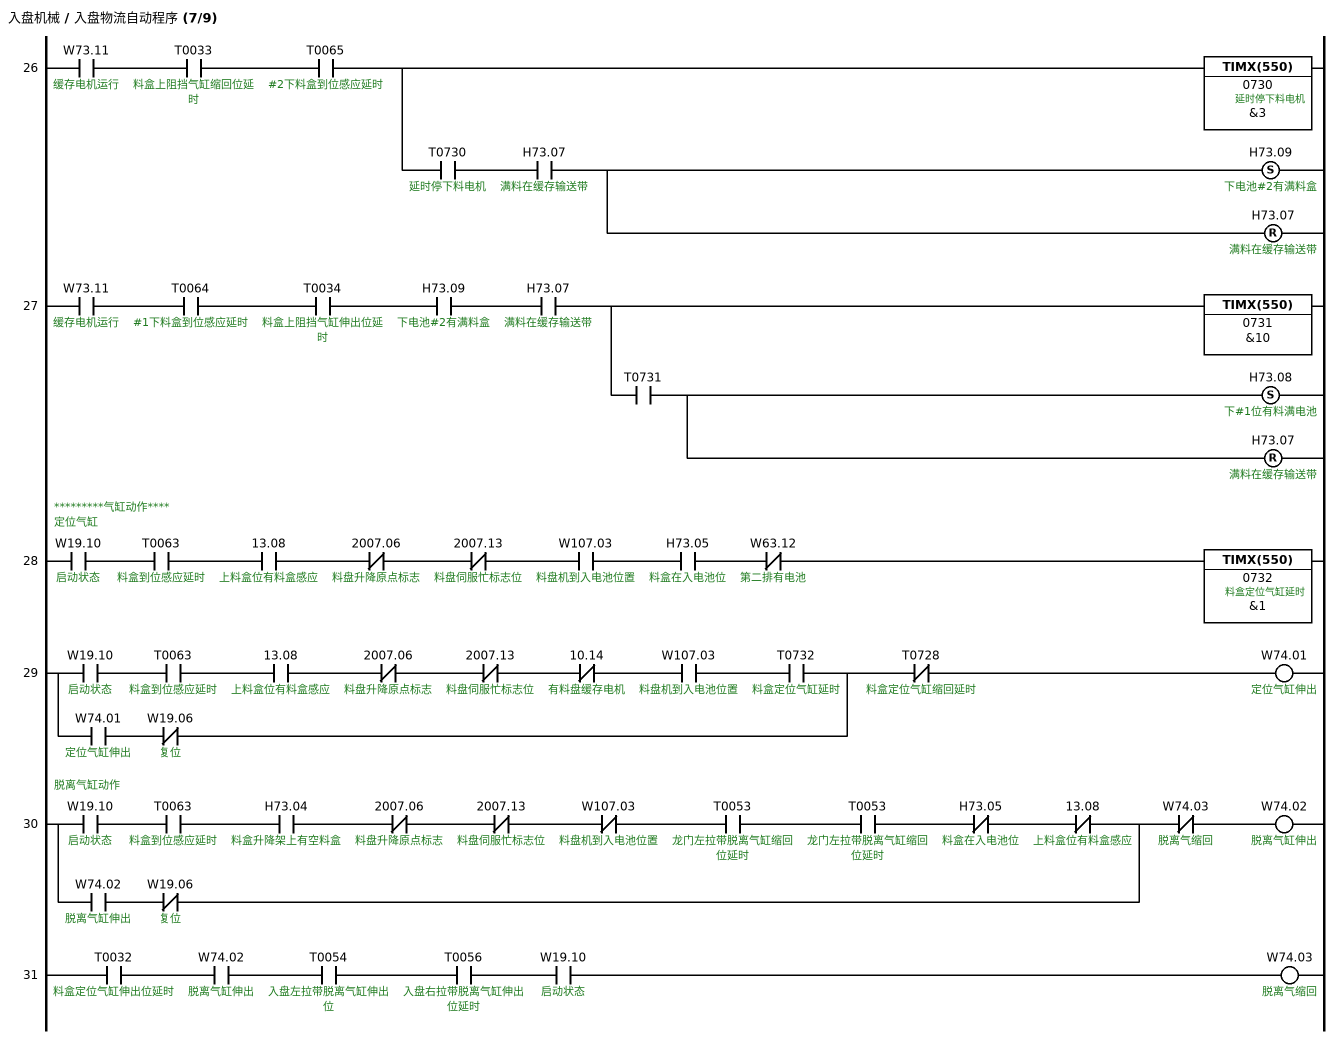
; rung 26
LD W73.11  ; 缓存电机运行
AND T0033  ; 料盒上阻挡气缸缩回位延时
AND T0065  ; #2下料盒到位感应延时
TIMX(550) 0730 &3  ; 延时停下料电机
AND T0730  ; 延时停下料电机
AND H73.07  ; 满料在缓存输送带
SET H73.09  ; 下电池#2有满料盒
RSET H73.07  ; 满料在缓存输送带
; rung 27
LD W73.11  ; 缓存电机运行
AND T0064  ; #1下料盒到位感应延时
AND T0034  ; 料盒上阻挡气缸伸出位延时
AND H73.09  ; 下电池#2有满料盒
AND H73.07  ; 满料在缓存输送带
TIMX(550) 0731 &10
AND T0731
SET H73.08  ; 下#1位有料满电池
RSET H73.07  ; 满料在缓存输送带
; rung 28: *********气缸动作**** / 定位气缸
LD W19.10  ; 启动状态
AND T0063  ; 料盒到位感应延时
AND 13.08  ; 上料盒位有料盒感应
ANDNOT 2007.06  ; 料盘升降原点标志
ANDNOT 2007.13  ; 料盘伺服忙标志位
AND W107.03  ; 料盘机到入电池位置
AND H73.05  ; 料盒在入电池位
ANDNOT W63.12  ; 第二排有电池
TIMX(550) 0732 &1  ; 料盒定位气缸延时
; rung 29
LD W19.10  ; 启动状态
AND T0063  ; 料盒到位感应延时
AND 13.08  ; 上料盒位有料盒感应
ANDNOT 2007.06  ; 料盘升降原点标志
ANDNOT 2007.13  ; 料盘伺服忙标志位
ANDNOT 10.14  ; 有料盘缓存电机
AND W107.03  ; 料盘机到入电池位置
AND T0732  ; 料盒定位气缸延时
LD W74.01  ; 定位气缸伸出
ANDNOT W19.06  ; 复位
ORLD
ANDNOT T0728  ; 料盒定位气缸缩回延时
OUT W74.01  ; 定位气缸伸出
; rung 30: 脱离气缸动作
LD W19.10  ; 启动状态
AND T0063  ; 料盒到位感应延时
AND H73.04  ; 料盒升降架上有空料盒
ANDNOT 2007.06  ; 料盘升降原点标志
ANDNOT 2007.13  ; 料盘伺服忙标志位
ANDNOT W107.03  ; 料盘机到入电池位置
AND T0053  ; 龙门左拉带脱离气缸缩回位延时
AND T0053  ; 龙门左拉带脱离气缸缩回位延时
ANDNOT H73.05  ; 料盒在入电池位
ANDNOT 13.08  ; 上料盒位有料盒感应
LD W74.02  ; 脱离气缸伸出
ANDNOT W19.06  ; 复位
ORLD
ANDNOT W74.03  ; 脱离气缩回
OUT W74.02  ; 脱离气缸伸出
; rung 31
LD T0032  ; 料盒定位气缸伸出位延时
AND W74.02  ; 脱离气缸伸出
AND T0054  ; 入盘左拉带脱离气缸伸出位
AND T0056  ; 入盘右拉带脱离气缸伸出位延时
AND W19.10  ; 启动状态
OUT W74.03  ; 脱离气缩回

